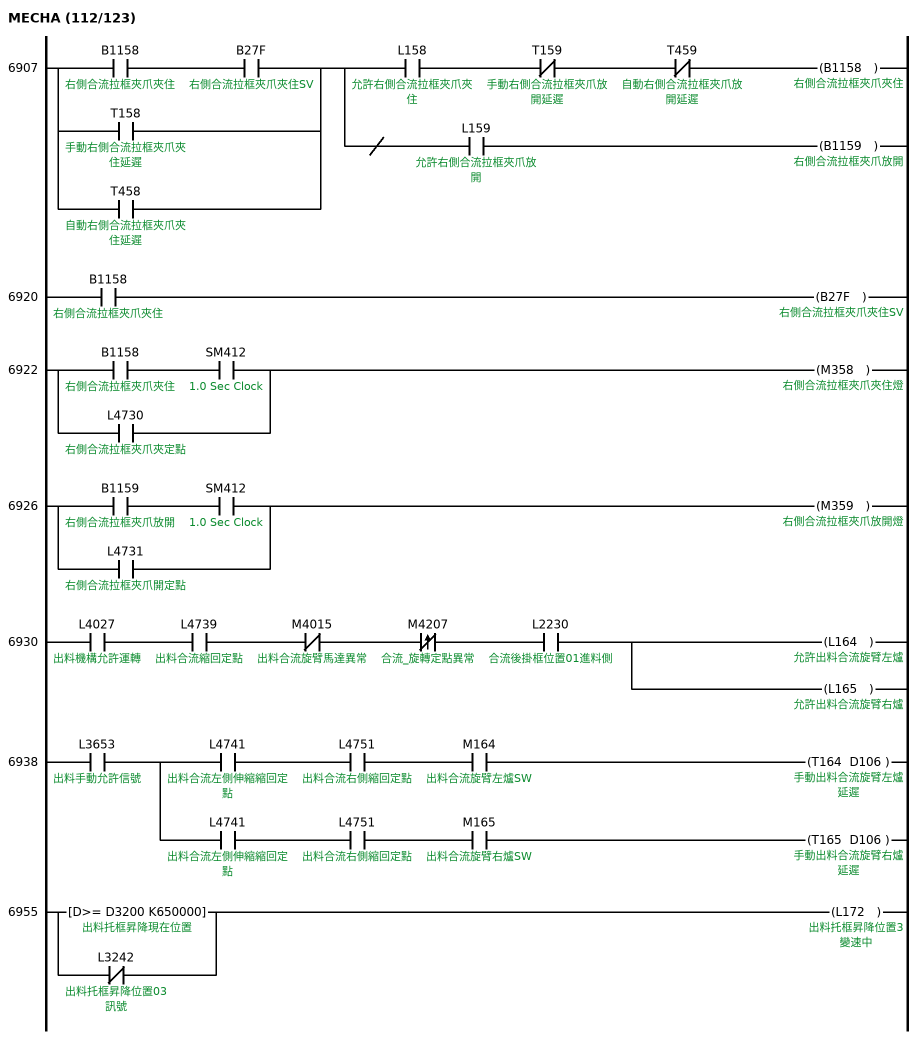
[picture p408: ladder of MECHA, rungs at steps 6907 to 6955]
6907  LD      B1158  ; 右側合流拉框夾爪夾住
      AND     B27F  ; 右側合流拉框夾爪夾住SV
      OR      T158  ; 手動右側合流拉框夾爪夾住延遲
      OR      T458  ; 自動右側合流拉框夾爪夾住延遲
      MPS
      AND     L158  ; 允許右側合流拉框夾爪夾住
      ANI     T159  ; 手動右側合流拉框夾爪放開延遲
      ANI     T459  ; 自動右側合流拉框夾爪放開延遲
      OUT     B1158  ; 右側合流拉框夾爪夾住
      MPP
      INV
      AND     L159  ; 允許右側合流拉框夾爪放開
      OUT     B1159  ; 右側合流拉框夾爪放開
6920  LD      B1158  ; 右側合流拉框夾爪夾住
      OUT     B27F  ; 右側合流拉框夾爪夾住SV
6922  LD      B1158  ; 右側合流拉框夾爪夾住
      AND     SM412  ; 1.0 Sec Clock
      OR      L4730  ; 右側合流拉框夾爪夾定點
      OUT     M358  ; 右側合流拉框夾爪夾住燈
6926  LD      B1159  ; 右側合流拉框夾爪放開
      AND     SM412  ; 1.0 Sec Clock
      OR      L4731  ; 右側合流拉框夾爪開定點
      OUT     M359  ; 右側合流拉框夾爪放開燈
6930  LD      L4027  ; 出料機構允許運轉
      AND     L4739  ; 出料合流縮回定點
      ANI     M4015  ; 出料合流旋臂馬達異常
      ANDPI   M4207  ; 合流_旋轉定點異常
      AND     L2230  ; 合流後掛框位置01進料側
      OUT     L164  ; 允許出料合流旋臂左爐
      OUT     L165  ; 允許出料合流旋臂右爐
6938  LD      L3653  ; 出料手動允許信號
      MPS
      AND     L4741  ; 出料合流左側伸縮縮回定點
      AND     L4751  ; 出料合流右側縮回定點
      AND     M164  ; 出料合流旋臂左爐SW
      OUT     T164 D106  ; 手動出料合流旋臂左爐延遲
      MPP
      AND     L4741  ; 出料合流左側伸縮縮回定點
      AND     L4751  ; 出料合流右側縮回定點
      AND     M165  ; 出料合流旋臂右爐SW
      OUT     T165 D106  ; 手動出料合流旋臂右爐延遲
6955  LDD>=   D3200 K650000  ; 出料托框昇降現在位置
      ORI     L3242  ; 出料托框昇降位置03 訊號
      OUT     L172  ; 出料托框昇降位置3 變速中
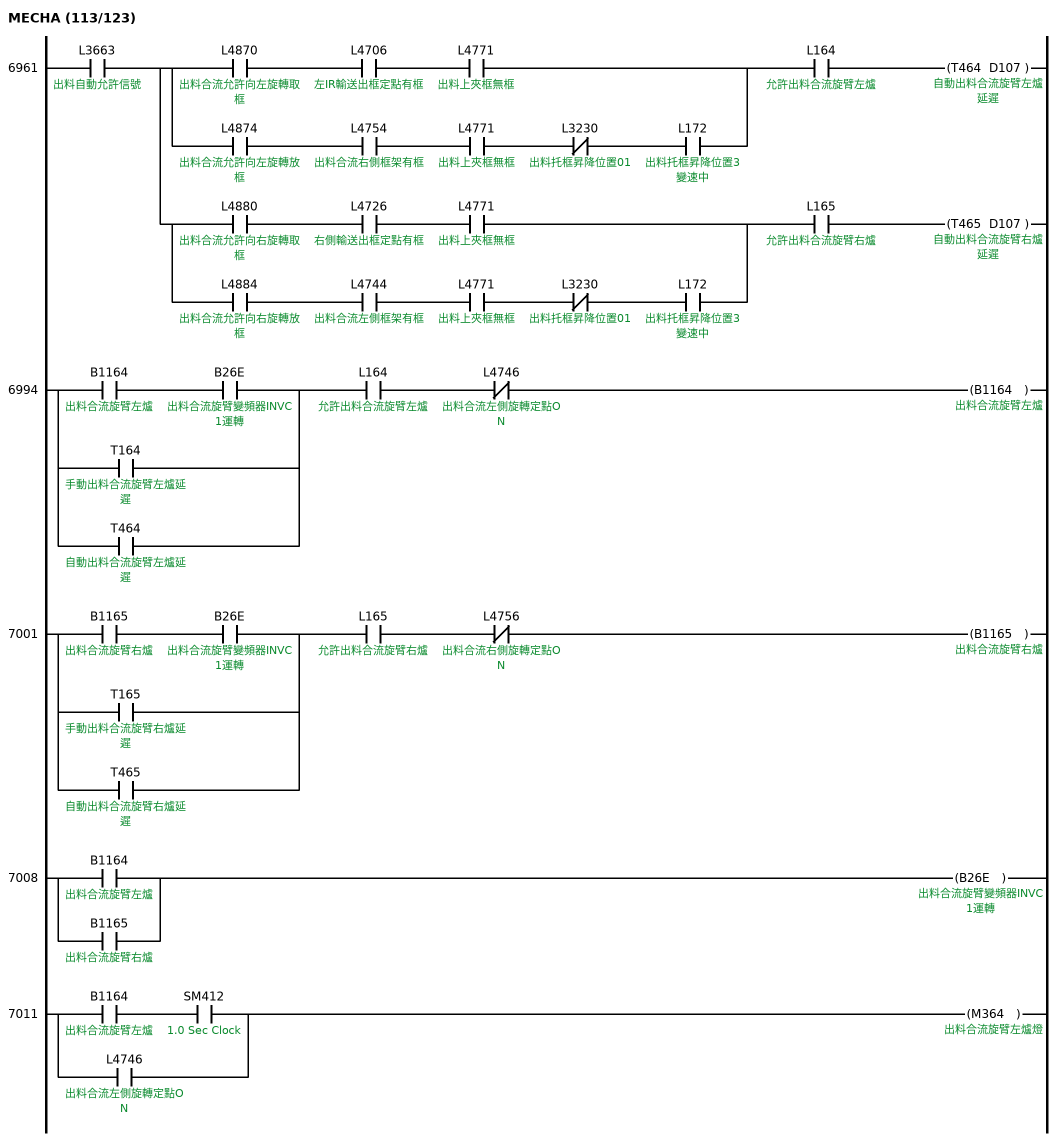
6961  LD      L3663  ; 出料自動允許信號
      MPS
      LD      L4870  ; 出料合流允許向左旋轉取框
      AND     L4706  ; 左IR輸送出框定點有框
      AND     L4771  ; 出料上夾框無框
      LD      L4874  ; 出料合流允許向左旋轉放框
      AND     L4754  ; 出料合流右側框架有框
      AND     L4771  ; 出料上夾框無框
      ANI     L3230  ; 出料托框昇降位置01
      AND     L172  ; 出料托框昇降位置3 變速中
      ORB
      ANB
      AND     L164  ; 允許出料合流旋臂左爐
      OUT     T464 D107  ; 自動出料合流旋臂左爐延遲
      MPP
      LD      L4880  ; 出料合流允許向右旋轉取框
      AND     L4726  ; 右側輸送出框定點有框
      AND     L4771  ; 出料上夾框無框
      LD      L4884  ; 出料合流允許向右旋轉放框
      AND     L4744  ; 出料合流左側框架有框
      AND     L4771  ; 出料上夾框無框
      ANI     L3230  ; 出料托框昇降位置01
      AND     L172  ; 出料托框昇降位置3 變速中
      ORB
      ANB
      AND     L165  ; 允許出料合流旋臂右爐
      OUT     T465 D107  ; 自動出料合流旋臂右爐延遲
6994  LD      B1164  ; 出料合流旋臂左爐
      AND     B26E  ; 出料合流旋臂變頻器INVC1運轉
      OR      T164  ; 手動出料合流旋臂左爐延遲
      OR      T464  ; 自動出料合流旋臂左爐延遲
      AND     L164  ; 允許出料合流旋臂左爐
      ANI     L4746  ; 出料合流左側旋轉定點ON
      OUT     B1164  ; 出料合流旋臂左爐
7001  LD      B1165  ; 出料合流旋臂右爐
      AND     B26E  ; 出料合流旋臂變頻器INVC1運轉
      OR      T165  ; 手動出料合流旋臂右爐延遲
      OR      T465  ; 自動出料合流旋臂右爐延遲
      AND     L165  ; 允許出料合流旋臂右爐
      ANI     L4756  ; 出料合流右側旋轉定點ON
      OUT     B1165  ; 出料合流旋臂右爐
7008  LD      B1164  ; 出料合流旋臂左爐
      OR      B1165  ; 出料合流旋臂右爐
      OUT     B26E  ; 出料合流旋臂變頻器INVC1運轉
7011  LD      B1164  ; 出料合流旋臂左爐
      AND     SM412  ; 1.0 Sec Clock
      OR      L4746  ; 出料合流左側旋轉定點ON
      OUT     M364  ; 出料合流旋臂左爐燈
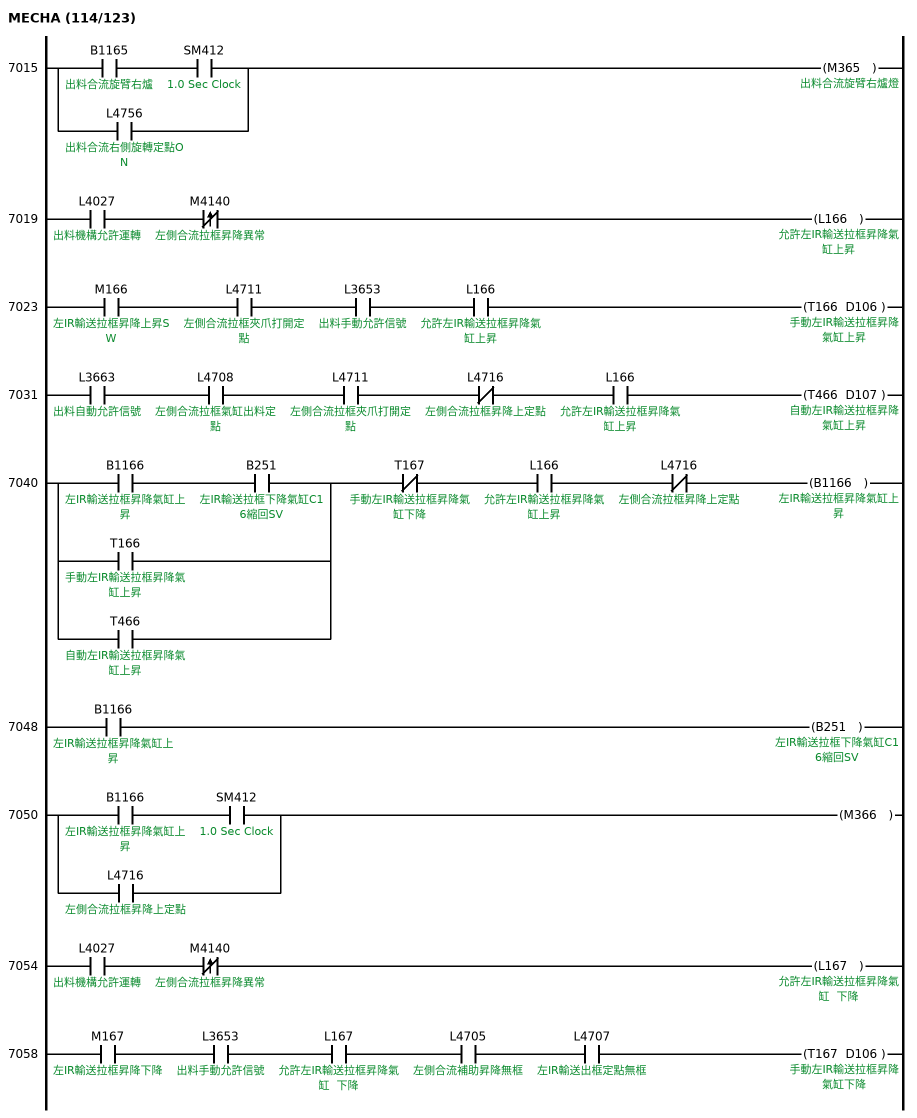
7015  LD      B1165  ; 出料合流旋臂右爐
      AND     SM412  ; 1.0 Sec Clock
      OR      L4756  ; 出料合流右側旋轉定點ON
      OUT     M365  ; 出料合流旋臂右爐燈
7019  LD      L4027  ; 出料機構允許運轉
      ANDPI   M4140  ; 左側合流拉框昇降異常
      OUT     L166  ; 允許左IR輸送拉框昇降氣缸上昇
7023  LD      M166  ; 左IR輸送拉框昇降上昇SW
      AND     L4711  ; 左側合流拉框夾爪打開定點
      AND     L3653  ; 出料手動允許信號
      AND     L166  ; 允許左IR輸送拉框昇降氣缸上昇
      OUT     T166 D106  ; 手動左IR輸送拉框昇降氣缸上昇
7031  LD      L3663  ; 出料自動允許信號
      AND     L4708  ; 左側合流拉框氣缸出料定點
      AND     L4711  ; 左側合流拉框夾爪打開定點
      ANI     L4716  ; 左側合流拉框昇降上定點
      AND     L166  ; 允許左IR輸送拉框昇降氣缸上昇
      OUT     T466 D107  ; 自動左IR輸送拉框昇降氣缸上昇
7040  LD      B1166  ; 左IR輸送拉框昇降氣缸上昇
      AND     B251  ; 左IR輸送拉框下降氣缸C16縮回SV
      OR      T166  ; 手動左IR輸送拉框昇降氣缸上昇
      OR      T466  ; 自動左IR輸送拉框昇降氣缸上昇
      ANI     T167  ; 手動左IR輸送拉框昇降氣缸下降
      AND     L166  ; 允許左IR輸送拉框昇降氣缸上昇
      ANI     L4716  ; 左側合流拉框昇降上定點
      OUT     B1166  ; 左IR輸送拉框昇降氣缸上昇
7048  LD      B1166  ; 左IR輸送拉框昇降氣缸上昇
      OUT     B251  ; 左IR輸送拉框下降氣缸C16縮回SV
7050  LD      B1166  ; 左IR輸送拉框昇降氣缸上昇
      AND     SM412  ; 1.0 Sec Clock
      OR      L4716  ; 左側合流拉框昇降上定點
      OUT     M366
7054  LD      L4027  ; 出料機構允許運轉
      ANDPI   M4140  ; 左側合流拉框昇降異常
      OUT     L167  ; 允許左IR輸送拉框昇降氣缸  下降
7058  LD      M167  ; 左IR輸送拉框昇降下降
      AND     L3653  ; 出料手動允許信號
      AND     L167  ; 允許左IR輸送拉框昇降氣缸  下降
      AND     L4705  ; 左側合流補助昇降無框
      AND     L4707  ; 左IR輸送出框定點無框
      OUT     T167 D106  ; 手動左IR輸送拉框昇降氣缸下降
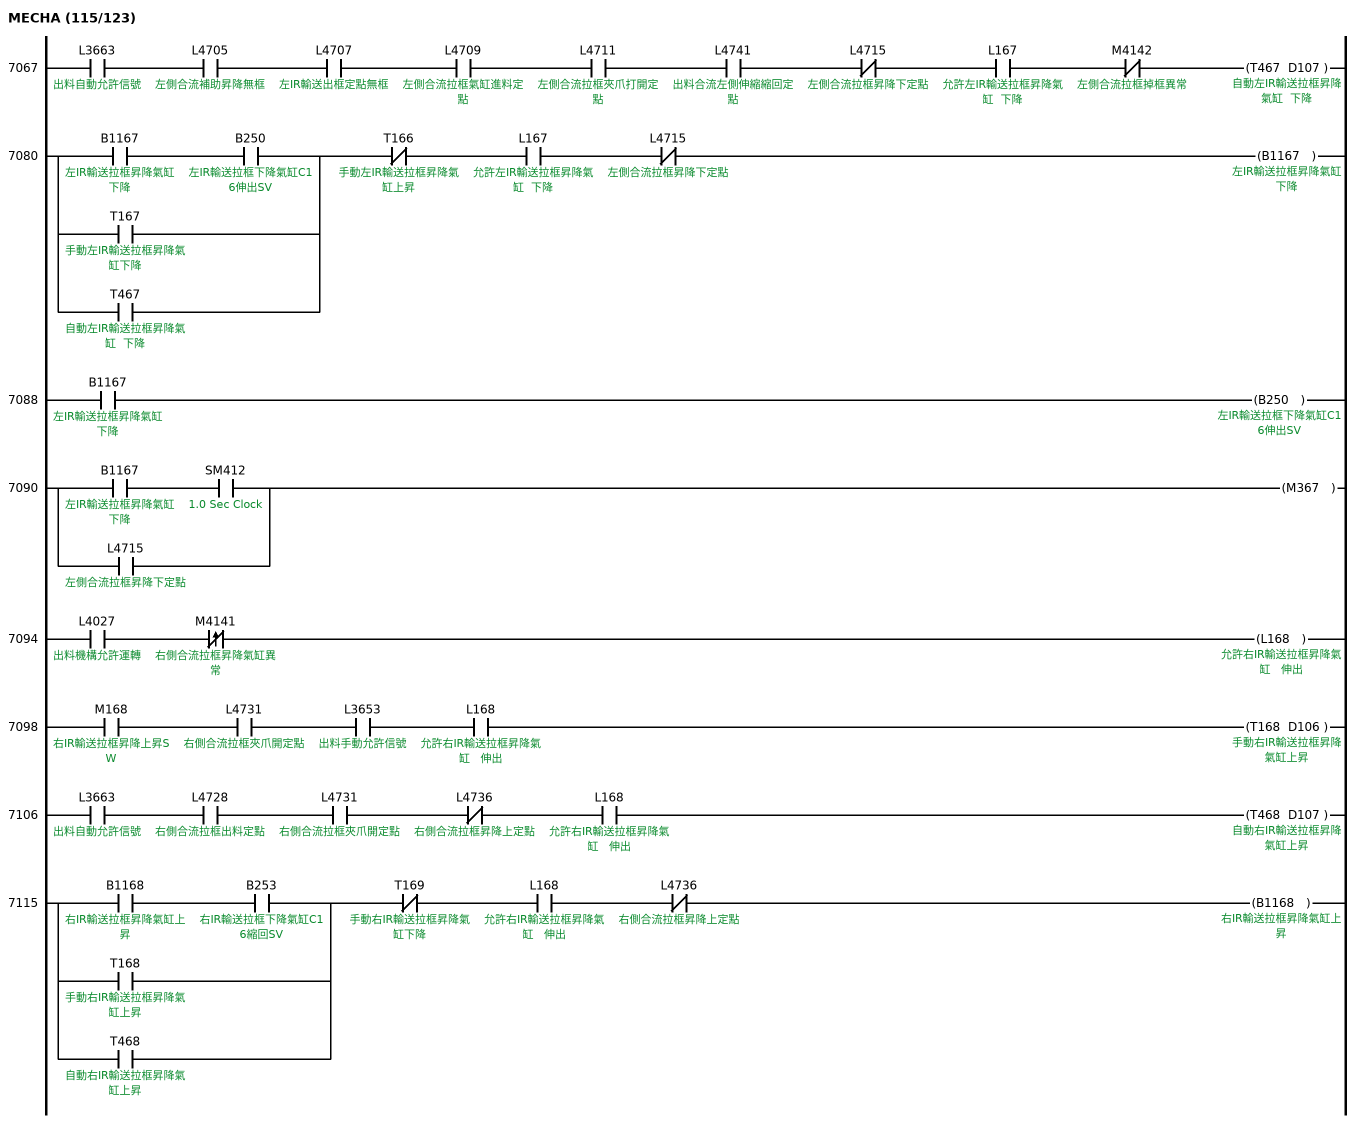
7067  LD      L3663  ; 出料自動允許信號
      AND     L4705  ; 左側合流補助昇降無框
      AND     L4707  ; 左IR輸送出框定點無框
      AND     L4709  ; 左側合流拉框氣缸進料定點
      AND     L4711  ; 左側合流拉框夾爪打開定點
      AND     L4741  ; 出料合流左側伸縮縮回定點
      ANI     L4715  ; 左側合流拉框昇降下定點
      AND     L167  ; 允許左IR輸送拉框昇降氣缸  下降
      ANI     M4142  ; 左側合流拉框掉框異常
      OUT     T467 D107  ; 自動左IR輸送拉框昇降氣缸  下降
7080  LD      B1167  ; 左IR輸送拉框昇降氣缸  下降
      AND     B250  ; 左IR輸送拉框下降氣缸C16伸出SV
      OR      T167  ; 手動左IR輸送拉框昇降氣缸下降
      OR      T467  ; 自動左IR輸送拉框昇降氣缸  下降
      ANI     T166  ; 手動左IR輸送拉框昇降氣缸上昇
      AND     L167  ; 允許左IR輸送拉框昇降氣缸  下降
      ANI     L4715  ; 左側合流拉框昇降下定點
      OUT     B1167  ; 左IR輸送拉框昇降氣缸  下降
7088  LD      B1167  ; 左IR輸送拉框昇降氣缸  下降
      OUT     B250  ; 左IR輸送拉框下降氣缸C16伸出SV
7090  LD      B1167  ; 左IR輸送拉框昇降氣缸  下降
      AND     SM412  ; 1.0 Sec Clock
      OR      L4715  ; 左側合流拉框昇降下定點
      OUT     M367
7094  LD      L4027  ; 出料機構允許運轉
      ANDPI   M4141  ; 右側合流拉框昇降氣缸異常
      OUT     L168  ; 允許右IR輸送拉框昇降氣缸   伸出
7098  LD      M168  ; 右IR輸送拉框昇降上昇SW
      AND     L4731  ; 右側合流拉框夾爪開定點
      AND     L3653  ; 出料手動允許信號
      AND     L168  ; 允許右IR輸送拉框昇降氣缸   伸出
      OUT     T168 D106  ; 手動右IR輸送拉框昇降氣缸上昇
7106  LD      L3663  ; 出料自動允許信號
      AND     L4728  ; 右側合流拉框出料定點
      AND     L4731  ; 右側合流拉框夾爪開定點
      ANI     L4736  ; 右側合流拉框昇降上定點
      AND     L168  ; 允許右IR輸送拉框昇降氣缸   伸出
      OUT     T468 D107  ; 自動右IR輸送拉框昇降氣缸上昇
7115  LD      B1168  ; 右IR輸送拉框昇降氣缸上昇
      AND     B253  ; 右IR輸送拉框下降氣缸C16縮回SV
      OR      T168  ; 手動右IR輸送拉框昇降氣缸上昇
      OR      T468  ; 自動右IR輸送拉框昇降氣缸上昇
      ANI     T169  ; 手動右IR輸送拉框昇降氣缸下降
      AND     L168  ; 允許右IR輸送拉框昇降氣缸   伸出
      ANI     L4736  ; 右側合流拉框昇降上定點
      OUT     B1168  ; 右IR輸送拉框昇降氣缸上昇
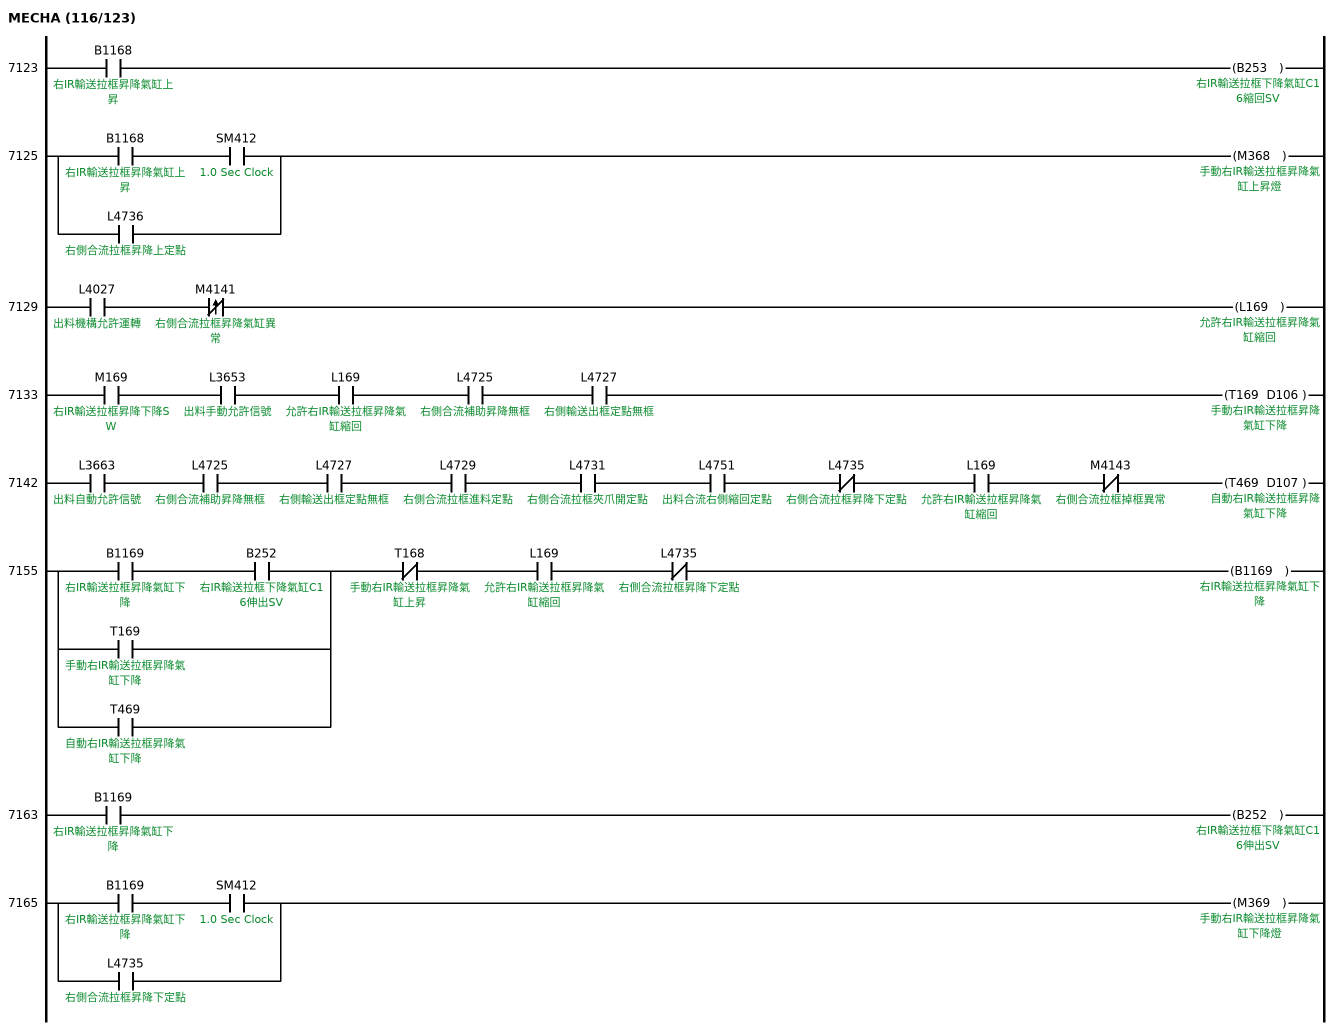
7123  LD      B1168  ; 右IR輸送拉框昇降氣缸上昇
      OUT     B253  ; 右IR輸送拉框下降氣缸C16縮回SV
7125  LD      B1168  ; 右IR輸送拉框昇降氣缸上昇
      AND     SM412  ; 1.0 Sec Clock
      OR      L4736  ; 右側合流拉框昇降上定點
      OUT     M368  ; 手動右IR輸送拉框昇降氣缸上昇燈
7129  LD      L4027  ; 出料機構允許運轉
      ANDPI   M4141  ; 右側合流拉框昇降氣缸異常
      OUT     L169  ; 允許右IR輸送拉框昇降氣缸縮回
7133  LD      M169  ; 右IR輸送拉框昇降下降SW
      AND     L3653  ; 出料手動允許信號
      AND     L169  ; 允許右IR輸送拉框昇降氣缸縮回
      AND     L4725  ; 右側合流補助昇降無框
      AND     L4727  ; 右側輸送出框定點無框
      OUT     T169 D106  ; 手動右IR輸送拉框昇降氣缸下降
7142  LD      L3663  ; 出料自動允許信號
      AND     L4725  ; 右側合流補助昇降無框
      AND     L4727  ; 右側輸送出框定點無框
      AND     L4729  ; 右側合流拉框進料定點
      AND     L4731  ; 右側合流拉框夾爪開定點
      AND     L4751  ; 出料合流右側縮回定點
      ANI     L4735  ; 右側合流拉框昇降下定點
      AND     L169  ; 允許右IR輸送拉框昇降氣缸縮回
      ANI     M4143  ; 右側合流拉框掉框異常
      OUT     T469 D107  ; 自動右IR輸送拉框昇降氣缸下降
7155  LD      B1169  ; 右IR輸送拉框昇降氣缸下降
      AND     B252  ; 右IR輸送拉框下降氣缸C16伸出SV
      OR      T169  ; 手動右IR輸送拉框昇降氣缸下降
      OR      T469  ; 自動右IR輸送拉框昇降氣缸下降
      ANI     T168  ; 手動右IR輸送拉框昇降氣缸上昇
      AND     L169  ; 允許右IR輸送拉框昇降氣缸縮回
      ANI     L4735  ; 右側合流拉框昇降下定點
      OUT     B1169  ; 右IR輸送拉框昇降氣缸下降
7163  LD      B1169  ; 右IR輸送拉框昇降氣缸下降
      OUT     B252  ; 右IR輸送拉框下降氣缸C16伸出SV
7165  LD      B1169  ; 右IR輸送拉框昇降氣缸下降
      AND     SM412  ; 1.0 Sec Clock
      OR      L4735  ; 右側合流拉框昇降下定點
      OUT     M369  ; 手動右IR輸送拉框昇降氣缸下降燈
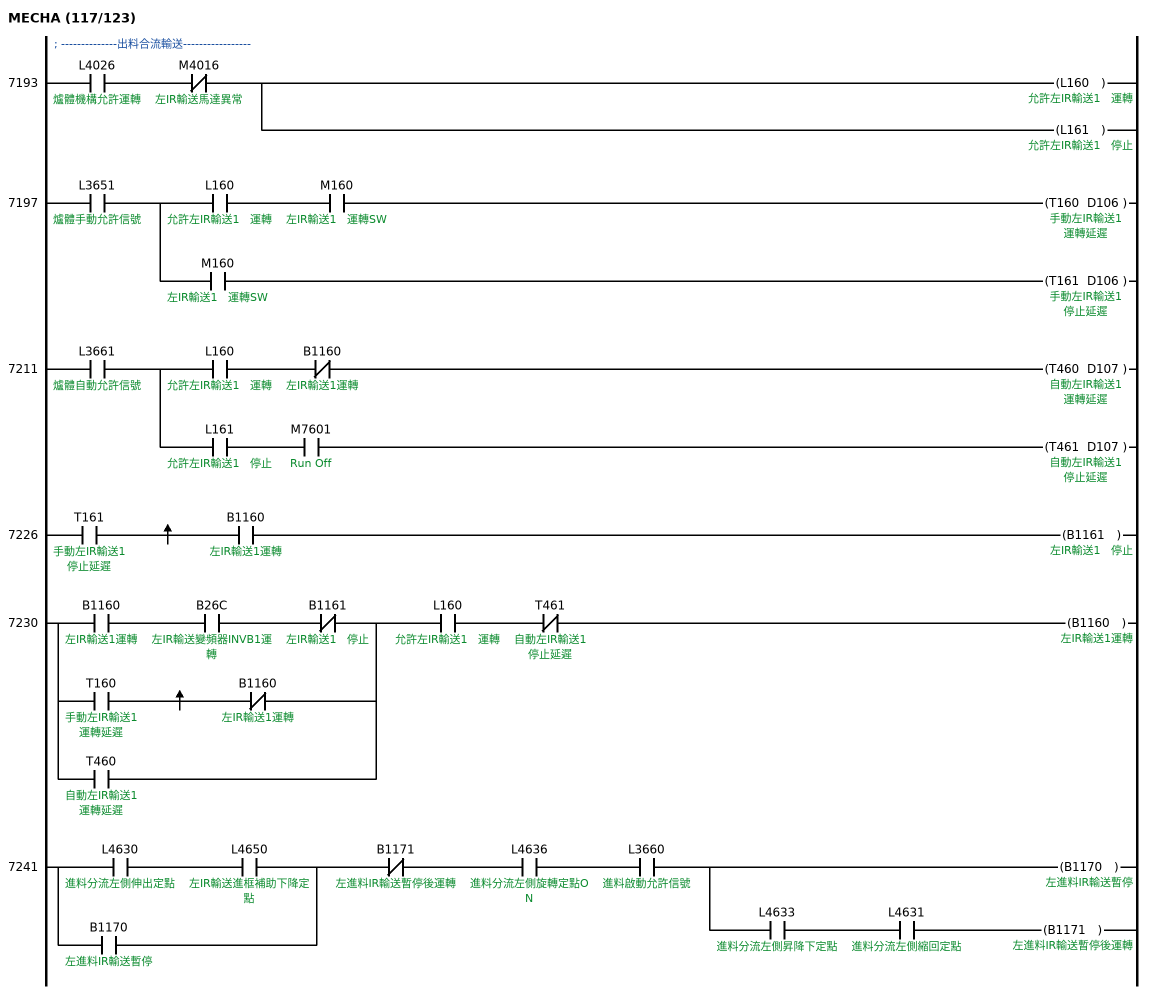
; --------------出料合流輸送-----------------
7193  LD      L4026  ; 爐體機構允許運轉
      ANI     M4016  ; 左IR輸送馬達異常
      OUT     L160  ; 允許左IR輸送1   運轉
      OUT     L161  ; 允許左IR輸送1   停止
7197  LD      L3651  ; 爐體手動允許信號
      MPS
      AND     L160  ; 允許左IR輸送1   運轉
      AND     M160  ; 左IR輸送1   運轉SW
      OUT     T160 D106  ; 手動左IR輸送1   運轉延遲
      MPP
      AND     M160  ; 左IR輸送1   運轉SW
      OUT     T161 D106  ; 手動左IR輸送1   停止延遲
7211  LD      L3661  ; 爐體自動允許信號
      MPS
      AND     L160  ; 允許左IR輸送1   運轉
      ANI     B1160  ; 左IR輸送1運轉
      OUT     T460 D107  ; 自動左IR輸送1   運轉延遲
      MPP
      AND     L161  ; 允許左IR輸送1   停止
      AND     M7601  ; Run Off
      OUT     T461 D107  ; 自動左IR輸送1   停止延遲
7226  LD      T161  ; 手動左IR輸送1   停止延遲
      MEP
      AND     B1160  ; 左IR輸送1運轉
      OUT     B1161  ; 左IR輸送1   停止
7230  LD      B1160  ; 左IR輸送1運轉
      AND     B26C  ; 左IR輸送變頻器INVB1運轉
      ANI     B1161  ; 左IR輸送1   停止
      LD      T160  ; 手動左IR輸送1   運轉延遲
      MEP
      ANI     B1160  ; 左IR輸送1運轉
      ORB
      OR      T460  ; 自動左IR輸送1   運轉延遲
      AND     L160  ; 允許左IR輸送1   運轉
      ANI     T461  ; 自動左IR輸送1   停止延遲
      OUT     B1160  ; 左IR輸送1運轉
7241  LD      L4630  ; 進料分流左側伸出定點
      AND     L4650  ; 左IR輸送進框補助下降定點
      OR      B1170  ; 左進料IR輸送暫停
      ANI     B1171  ; 左進料IR輸送暫停後運轉
      AND     L4636  ; 進料分流左側旋轉定點ON
      AND     L3660  ; 進料啟動允許信號
      OUT     B1170  ; 左進料IR輸送暫停
      AND     L4633  ; 進料分流左側昇降下定點
      AND     L4631  ; 進料分流左側縮回定點
      OUT     B1171  ; 左進料IR輸送暫停後運轉
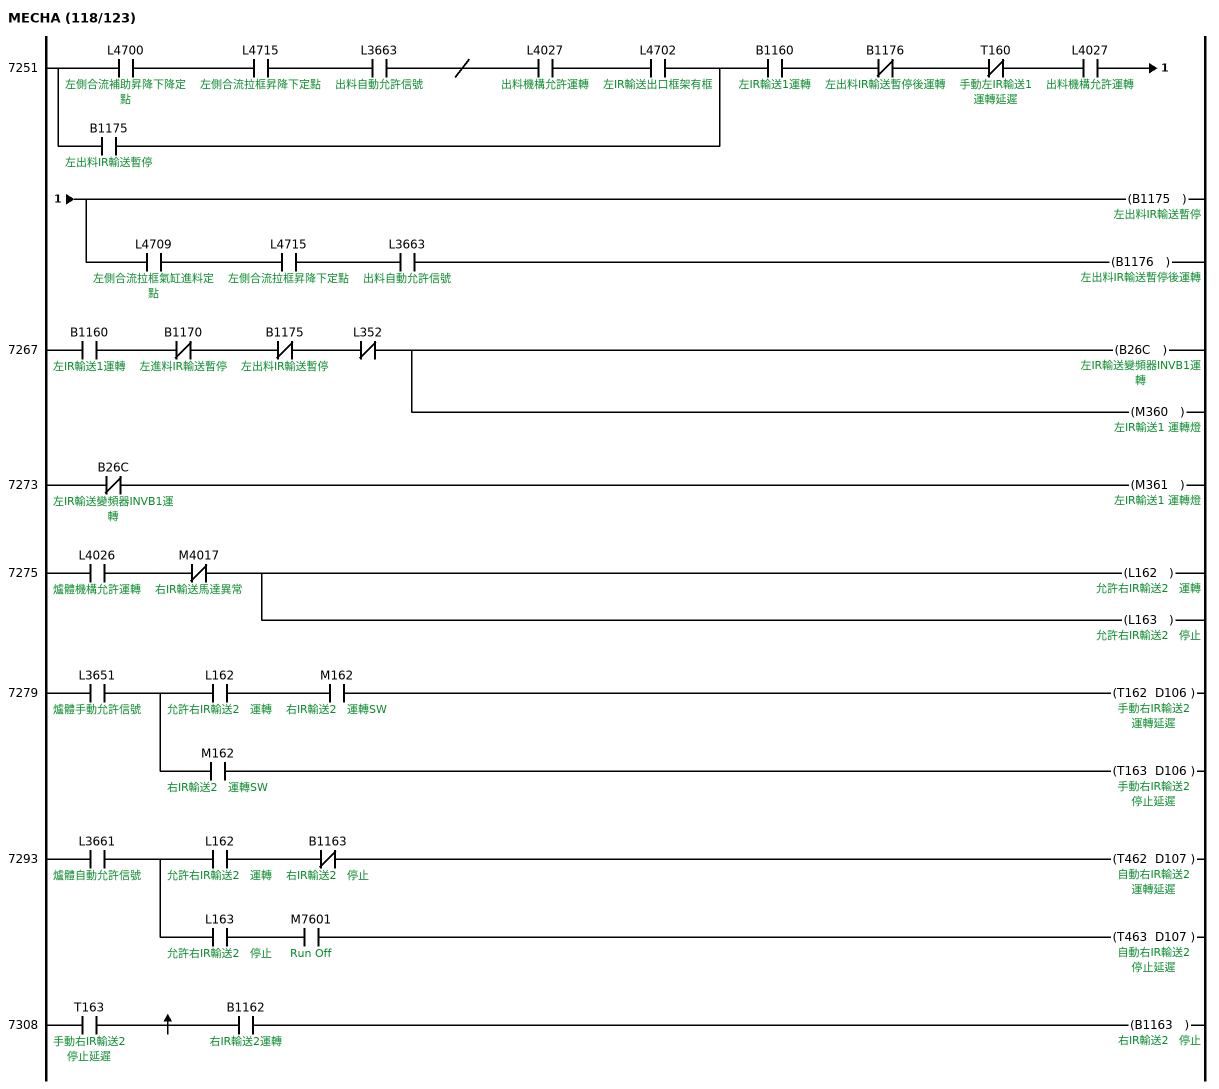
7251  LD      L4700  ; 左側合流補助昇降下降定點
      AND     L4715  ; 左側合流拉框昇降下定點
      AND     L3663  ; 出料自動允許信號
      INV
      AND     L4027  ; 出料機構允許運轉
      AND     L4702  ; 左IR輸送出口框架有框
      OR      B1175  ; 左出料IR輸送暫停
      AND     B1160  ; 左IR輸送1運轉
      ANI     B1176  ; 左出料IR輸送暫停後運轉
      ANI     T160  ; 手動左IR輸送1   運轉延遲
      AND     L4027  ; 出料機構允許運轉
      OUT     B1175  ; 左出料IR輸送暫停
      AND     L4709  ; 左側合流拉框氣缸進料定點
      AND     L4715  ; 左側合流拉框昇降下定點
      AND     L3663  ; 出料自動允許信號
      OUT     B1176  ; 左出料IR輸送暫停後運轉
7267  LD      B1160  ; 左IR輸送1運轉
      ANI     B1170  ; 左進料IR輸送暫停
      ANI     B1175  ; 左出料IR輸送暫停
      ANI     L352
      OUT     B26C  ; 左IR輸送變頻器INVB1運轉
      OUT     M360  ; 左IR輸送1 運轉燈
7273  LDI     B26C  ; 左IR輸送變頻器INVB1運轉
      OUT     M361  ; 左IR輸送1 運轉燈
7275  LD      L4026  ; 爐體機構允許運轉
      ANI     M4017  ; 右IR輸送馬達異常
      OUT     L162  ; 允許右IR輸送2   運轉
      OUT     L163  ; 允許右IR輸送2   停止
7279  LD      L3651  ; 爐體手動允許信號
      MPS
      AND     L162  ; 允許右IR輸送2   運轉
      AND     M162  ; 右IR輸送2   運轉SW
      OUT     T162 D106  ; 手動右IR輸送2   運轉延遲
      MPP
      AND     M162  ; 右IR輸送2   運轉SW
      OUT     T163 D106  ; 手動右IR輸送2   停止延遲
7293  LD      L3661  ; 爐體自動允許信號
      MPS
      AND     L162  ; 允許右IR輸送2   運轉
      ANI     B1163  ; 右IR輸送2   停止
      OUT     T462 D107  ; 自動右IR輸送2   運轉延遲
      MPP
      AND     L163  ; 允許右IR輸送2   停止
      AND     M7601  ; Run Off
      OUT     T463 D107  ; 自動右IR輸送2   停止延遲
7308  LD      T163  ; 手動右IR輸送2   停止延遲
      MEP
      AND     B1162  ; 右IR輸送2運轉
      OUT     B1163  ; 右IR輸送2   停止
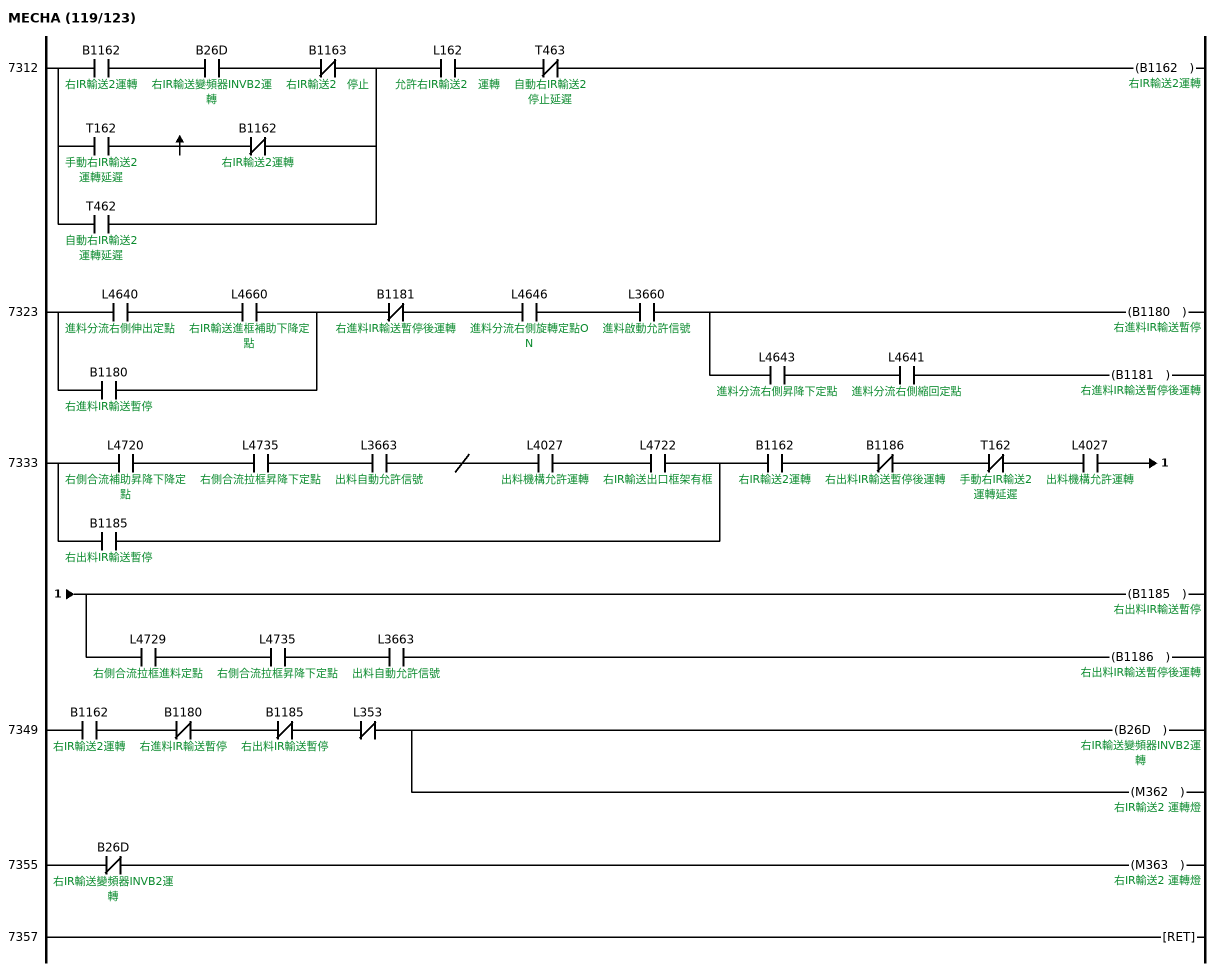
7312  LD      B1162  ; 右IR輸送2運轉
      AND     B26D  ; 右IR輸送變頻器INVB2運轉
      ANI     B1163  ; 右IR輸送2   停止
      LD      T162  ; 手動右IR輸送2   運轉延遲
      MEP
      ANI     B1162  ; 右IR輸送2運轉
      ORB
      OR      T462  ; 自動右IR輸送2   運轉延遲
      AND     L162  ; 允許右IR輸送2   運轉
      ANI     T463  ; 自動右IR輸送2   停止延遲
      OUT     B1162  ; 右IR輸送2運轉
7323  LD      L4640  ; 進料分流右側伸出定點
      AND     L4660  ; 右IR輸送進框補助下降定點
      OR      B1180  ; 右進料IR輸送暫停
      ANI     B1181  ; 右進料IR輸送暫停後運轉
      AND     L4646  ; 進料分流右側旋轉定點ON
      AND     L3660  ; 進料啟動允許信號
      OUT     B1180  ; 右進料IR輸送暫停
      AND     L4643  ; 進料分流右側昇降下定點
      AND     L4641  ; 進料分流右側縮回定點
      OUT     B1181  ; 右進料IR輸送暫停後運轉
7333  LD      L4720  ; 右側合流補助昇降下降定點
      AND     L4735  ; 右側合流拉框昇降下定點
      AND     L3663  ; 出料自動允許信號
      INV
      AND     L4027  ; 出料機構允許運轉
      AND     L4722  ; 右IR輸送出口框架有框
      OR      B1185  ; 右出料IR輸送暫停
      AND     B1162  ; 右IR輸送2運轉
      ANI     B1186  ; 右出料IR輸送暫停後運轉
      ANI     T162  ; 手動右IR輸送2   運轉延遲
      AND     L4027  ; 出料機構允許運轉
      OUT     B1185  ; 右出料IR輸送暫停
      AND     L4729  ; 右側合流拉框進料定點
      AND     L4735  ; 右側合流拉框昇降下定點
      AND     L3663  ; 出料自動允許信號
      OUT     B1186  ; 右出料IR輸送暫停後運轉
7349  LD      B1162  ; 右IR輸送2運轉
      ANI     B1180  ; 右進料IR輸送暫停
      ANI     B1185  ; 右出料IR輸送暫停
      ANI     L353
      OUT     B26D  ; 右IR輸送變頻器INVB2運轉
      OUT     M362  ; 右IR輸送2 運轉燈
7355  LDI     B26D  ; 右IR輸送變頻器INVB2運轉
      OUT     M363  ; 右IR輸送2 運轉燈
7357  RET
      P1071
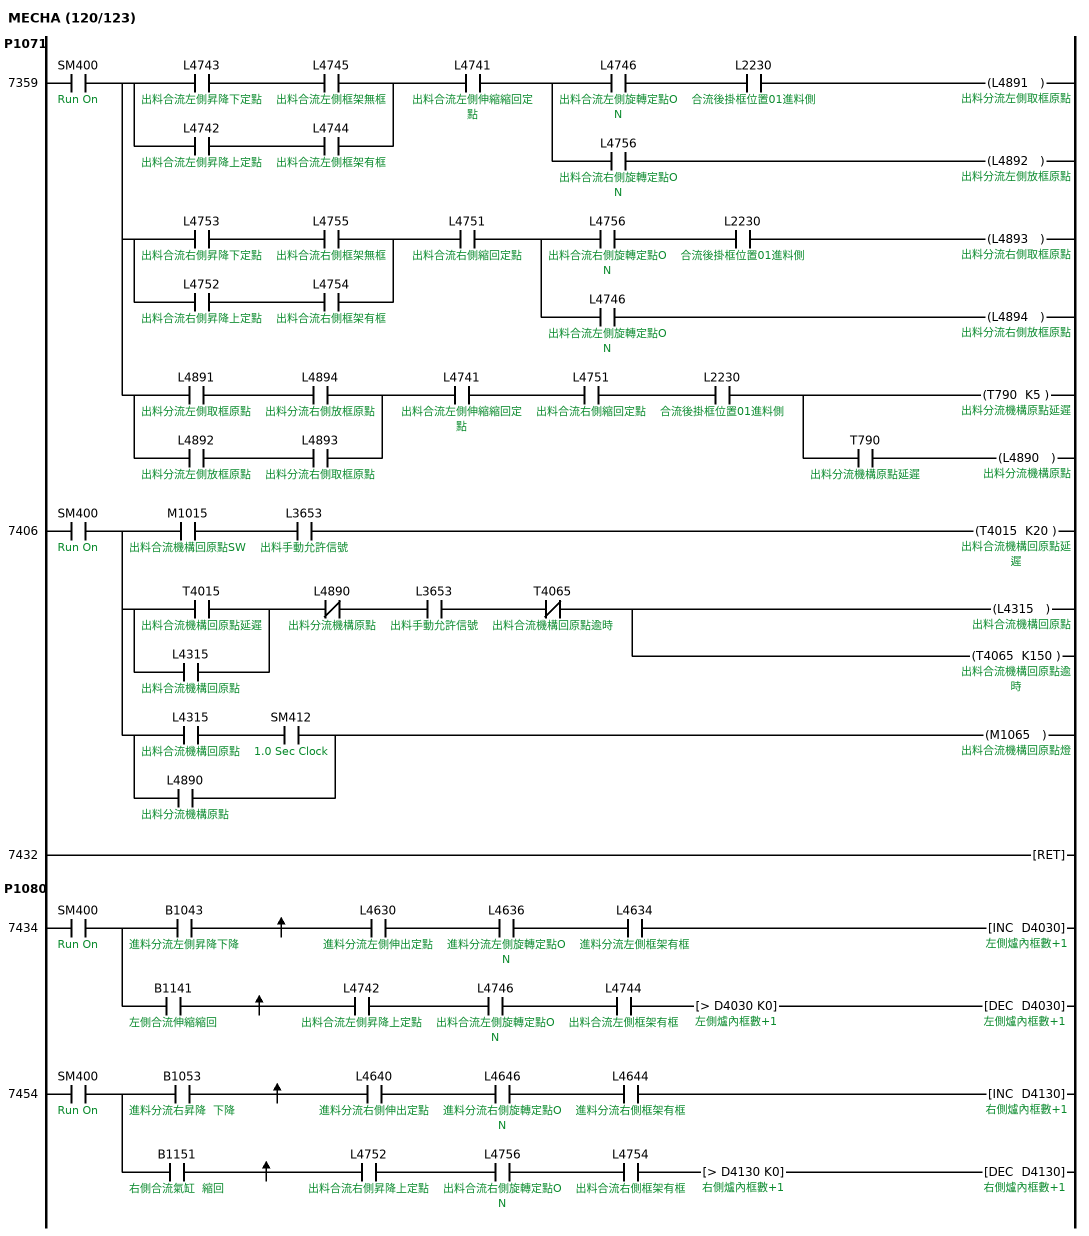
7359  LD      SM400  ; Run On
      MPS
      LD      L4743  ; 出料合流左側昇降下定點
      AND     L4745  ; 出料合流左側框架無框
      LD      L4742  ; 出料合流左側昇降上定點
      AND     L4744  ; 出料合流左側框架有框
      ORB
      ANB
      AND     L4741  ; 出料合流左側伸縮縮回定點
      MPS
      AND     L4746  ; 出料合流左側旋轉定點ON
      AND     L2230  ; 合流後掛框位置01進料側
      OUT     L4891  ; 出料分流左側取框原點
      MPP
      AND     L4756  ; 出料合流右側旋轉定點ON
      OUT     L4892  ; 出料分流左側放框原點
      MRD
      LD      L4753  ; 出料合流右側昇降下定點
      AND     L4755  ; 出料合流右側框架無框
      LD      L4752  ; 出料合流右側昇降上定點
      AND     L4754  ; 出料合流右側框架有框
      ORB
      ANB
      AND     L4751  ; 出料合流右側縮回定點
      MPS
      AND     L4756  ; 出料合流右側旋轉定點ON
      AND     L2230  ; 合流後掛框位置01進料側
      OUT     L4893  ; 出料分流右側取框原點
      MPP
      AND     L4746  ; 出料合流左側旋轉定點ON
      OUT     L4894  ; 出料分流右側放框原點
      MPP
      LD      L4891  ; 出料分流左側取框原點
      AND     L4894  ; 出料分流右側放框原點
      LD      L4892  ; 出料分流左側放框原點
      AND     L4893  ; 出料分流右側取框原點
      ORB
      ANB
      AND     L4741  ; 出料合流左側伸縮縮回定點
      AND     L4751  ; 出料合流右側縮回定點
      AND     L2230  ; 合流後掛框位置01進料側
      OUT     T790 K5  ; 出料分流機構原點延遲
      AND     T790  ; 出料分流機構原點延遲
      OUT     L4890  ; 出料分流機構原點
7406  LD      SM400  ; Run On
      MPS
      AND     M1015  ; 出料合流機構回原點SW
      AND     L3653  ; 出料手動允許信號
      OUT     T4015 K20  ; 出料合流機構回原點延遲
      MRD
      LD      T4015  ; 出料合流機構回原點延遲
      OR      L4315  ; 出料合流機構回原點
      ANB
      ANI     L4890  ; 出料分流機構原點
      AND     L3653  ; 出料手動允許信號
      ANI     T4065  ; 出料合流機構回原點逾時
      OUT     L4315  ; 出料合流機構回原點
      OUT     T4065 K150  ; 出料合流機構回原點逾時
      MPP
      LD      L4315  ; 出料合流機構回原點
      AND     SM412  ; 1.0 Sec Clock
      OR      L4890  ; 出料分流機構原點
      ANB
      OUT     M1065  ; 出料合流機構回原點燈
7432  RET
      P1080
7434  LD      SM400  ; Run On
      MPS
      AND     B1043  ; 進料分流左側昇降下降
      MEP
      AND     L4630  ; 進料分流左側伸出定點
      AND     L4636  ; 進料分流左側旋轉定點ON
      AND     L4634  ; 進料分流左側框架有框
      INC     D4030  ; 左側爐內框數+1
      MPP
      AND     B1141  ; 左側合流伸縮縮回
      MEP
      AND     L4742  ; 出料合流左側昇降上定點
      AND     L4746  ; 出料合流左側旋轉定點ON
      AND     L4744  ; 出料合流左側框架有框
      AND>    D4030 K0  ; 左側爐內框數+1
      DEC     D4030
7454  LD      SM400  ; Run On
      MPS
      AND     B1053  ; 進料分流右昇降  下降
      MEP
      AND     L4640  ; 進料分流右側伸出定點
      AND     L4646  ; 進料分流右側旋轉定點ON
      AND     L4644  ; 進料分流右側框架有框
      INC     D4130  ; 右側爐內框數+1
      MPP
      AND     B1151  ; 右側合流氣缸  縮回
      MEP
      AND     L4752  ; 出料合流右側昇降上定點
      AND     L4756  ; 出料合流右側旋轉定點ON
      AND     L4754  ; 出料合流右側框架有框
      AND>    D4130 K0  ; 右側爐內框數+1
      DEC     D4130
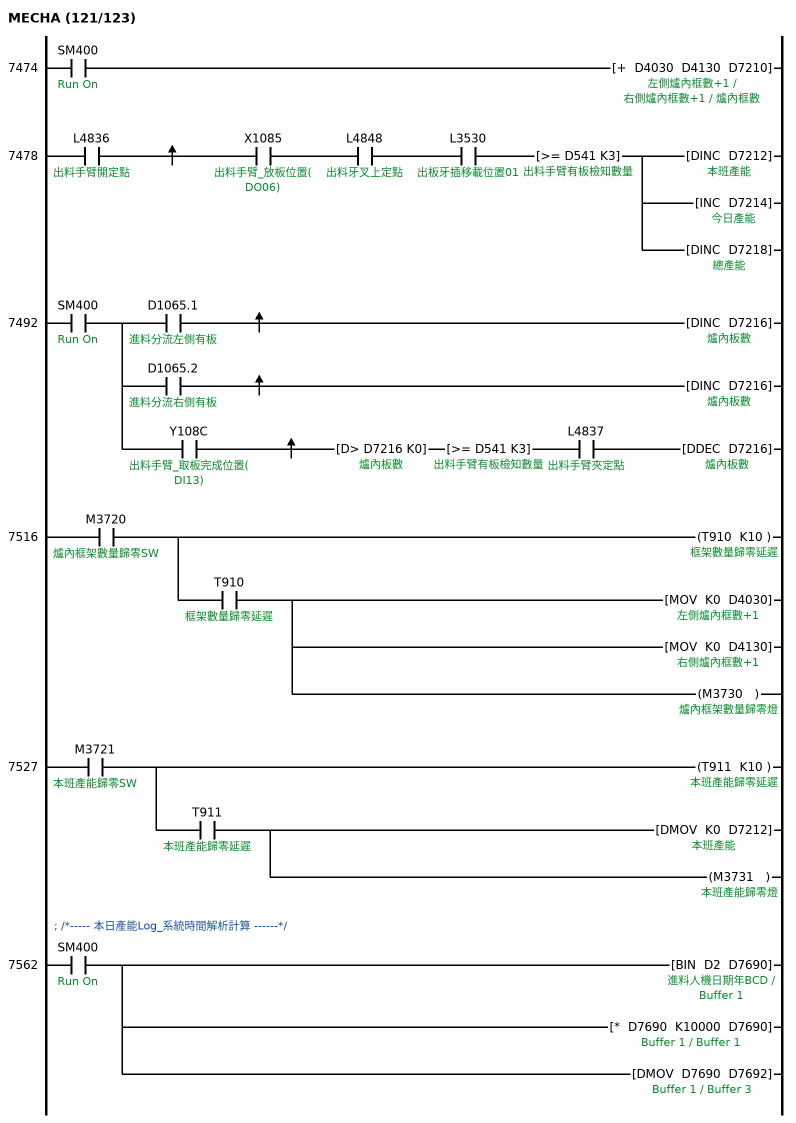
7474  LD      SM400  ; Run On
      +       D4030 D4130 D7210  ; 爐內框數
7478  LD      L4836  ; 出料手臂開定點
      MEP
      AND     X1085  ; 出料手臂_放板位置(DO06)
      AND     L4848  ; 出料牙叉上定點
      AND     L3530  ; 出板牙插移載位置01
      AND>=   D541 K3  ; 出料手臂有板檢知數量
      DINC    D7212  ; 本班產能
      INC     D7214  ; 今日產能
      DINC    D7218  ; 總產能
7492  LD      SM400  ; Run On
      MPS
      AND     D1065.1  ; 進料分流左側有板
      MEP
      DINC    D7216  ; 爐內板數
      MRD
      AND     D1065.2  ; 進料分流右側有板
      MEP
      DINC    D7216
      MPP
      AND     Y108C  ; 出料手臂_取板完成位置(DI13)
      MEP
      ANDD>   D7216 K0  ; 爐內板數
      AND>=   D541 K3  ; 出料手臂有板檢知數量
      AND     L4837  ; 出料手臂夾定點
      DDEC    D7216
7516  LD      M3720  ; 爐內框架數量歸零SW
      OUT     T910 K10  ; 框架數量歸零延遲
      AND     T910  ; 框架數量歸零延遲
      MOV     K0 D4030
      MOV     K0 D4130
      OUT     M3730  ; 爐內框架數量歸零燈
7527  LD      M3721  ; 本班產能歸零SW
      OUT     T911 K10  ; 本班產能歸零延遲
      AND     T911  ; 本班產能歸零延遲
      DMOV    K0 D7212
      OUT     M3731  ; 本班產能歸零燈
; /*----- 本日產能Log_系統時間解析計算 ------*/
7562  LD      SM400  ; Run On
      BIN     D2 D7690  ; 進料人機日期年BCD / Buffer 1
      *       D7690 K10000 D7690
      DMOV    D7690 D7692  ; Buffer 3
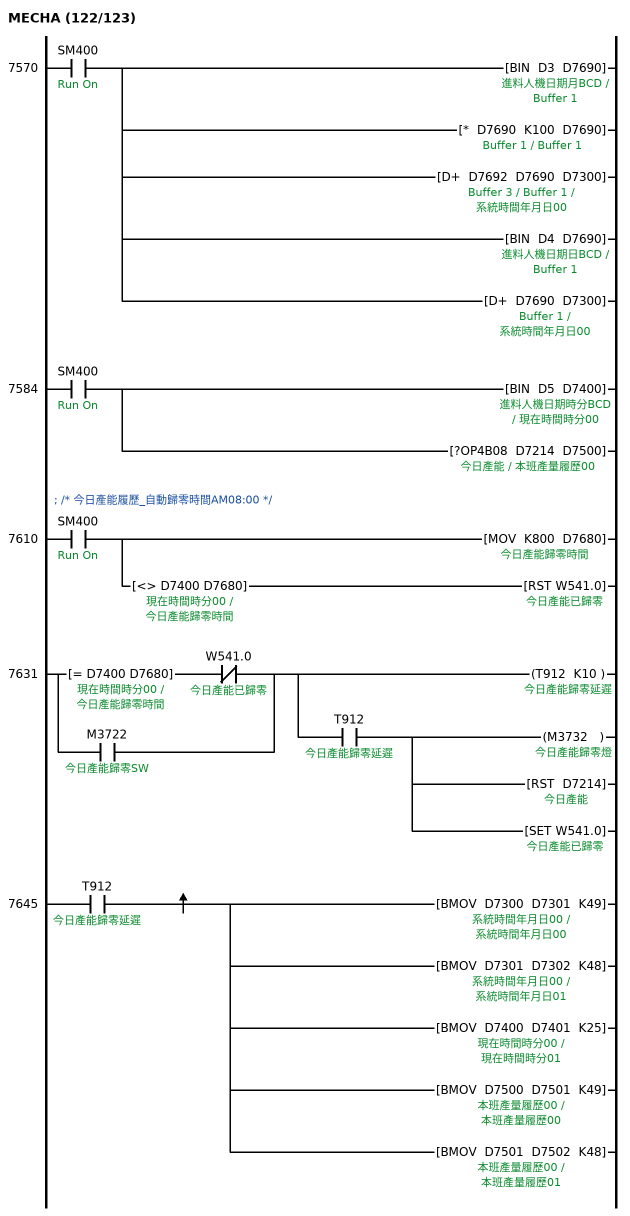
7570  LD      SM400  ; Run On
      BIN     D3 D7690  ; 進料人機日期月BCD
      *       D7690 K100 D7690
      D+      D7692 D7690 D7300  ; 系統時間年月日00
      BIN     D4 D7690  ; 進料人機日期日BCD
      D+      D7690 D7300
7584  LD      SM400  ; Run On
      BIN     D5 D7400  ; 進料人機日期時分BCD / 現在時間時分00
      ?OP4B08 D7214 D7500  ; 本班產量履歷00
; /* 今日產能履歷_自動歸零時間AM08:00 */
7610  LD      SM400  ; Run On
      MOV     K800 D7680  ; 今日產能歸零時間
        [note] 今日產能歸零時間_AM08:00
      AND<>   D7400 D7680  ; 現在時間時分00 / 今日產能歸零時間
      RST     W541.0  ; 今日產能已歸零
7631  LD=     D7400 D7680  ; 現在時間時分00 / 今日產能歸零時間
      ANI     W541.0  ; 今日產能已歸零
      OR      M3722  ; 今日產能歸零SW
      OUT     T912 K10  ; 今日產能歸零延遲
      AND     T912  ; 今日產能歸零延遲
      OUT     M3732  ; 今日產能歸零燈
      RST     D7214  ; 今日產能
      SET     W541.0  ; 今日產能已歸零
7645  LD      T912  ; 今日產能歸零延遲
      MEP
      BMOV    D7300 D7301 K49  ; 系統時間年月日00
      BMOV    D7301 D7302 K48  ; 系統時間年月日01
      BMOV    D7400 D7401 K25  ; 現在時間時分01
      BMOV    D7500 D7501 K49  ; 本班產量履歷00
      BMOV    D7501 D7502 K48  ; 本班產量履歷01
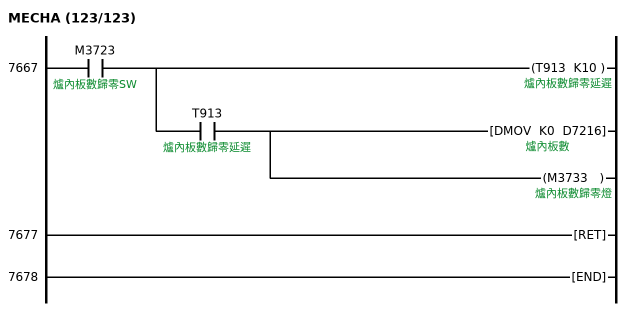
7667  LD      M3723  ; 爐內板數歸零SW
      OUT     T913 K10  ; 爐內板數歸零延遲
      AND     T913  ; 爐內板數歸零延遲
      DMOV    K0 D7216
      OUT     M3733  ; 爐內板數歸零燈
7677  RET
7678  END
END_PROGRAM

PROGRAM ORIGIN
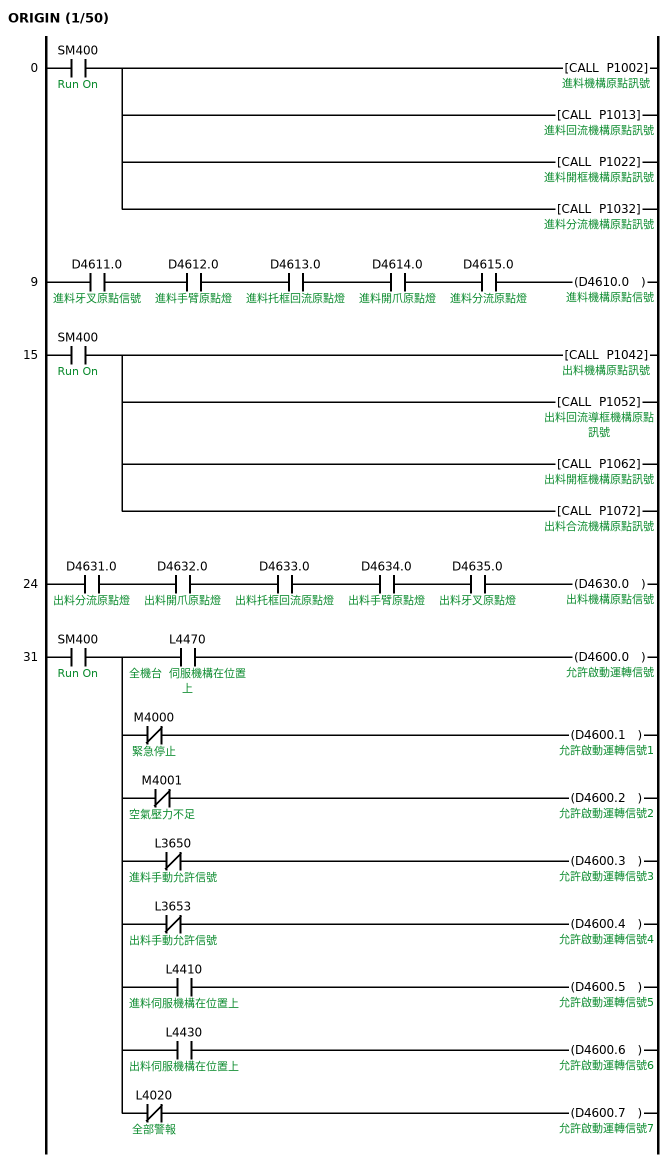
0     LD      SM400  ; Run On
      CALL    P1002  ; 進料機構原點訊號
      CALL    P1013  ; 進料回流機構原點訊號
      CALL    P1022  ; 進料開框機構原點訊號
      CALL    P1032  ; 進料分流機構原點訊號
9     LD      D4611.0  ; 進料牙叉原點信號
      AND     D4612.0  ; 進料手臂原點燈
      AND     D4613.0  ; 進料托框回流原點燈
      AND     D4614.0  ; 進料開爪原點燈
      AND     D4615.0  ; 進料分流原點燈
      OUT     D4610.0  ; 進料機構原點信號
15    LD      SM400  ; Run On
      CALL    P1042  ; 出料機構原點訊號
      CALL    P1052  ; 出料回流導框機構原點訊號
      CALL    P1062  ; 出料開框機構原點訊號
      CALL    P1072  ; 出料合流機構原點訊號
24    LD      D4631.0  ; 出料分流原點燈
      AND     D4632.0  ; 出料開爪原點燈
      AND     D4633.0  ; 出料托框回流原點燈
      AND     D4634.0  ; 出料手臂原點燈
      AND     D4635.0  ; 出料牙叉原點燈
      OUT     D4630.0  ; 出料機構原點信號
31    LD      SM400  ; Run On
      MPS
      AND     L4470  ; 全機台  伺服機構在位置上
      OUT     D4600.0  ; 允許啟動運轉信號
      MRD
      ANI     M4000  ; 緊急停止
      OUT     D4600.1  ; 允許啟動運轉信號1
      MRD
      ANI     M4001  ; 空氣壓力不足
      OUT     D4600.2  ; 允許啟動運轉信號2
      MRD
      ANI     L3650  ; 進料手動允許信號
      OUT     D4600.3  ; 允許啟動運轉信號3
      MRD
      ANI     L3653  ; 出料手動允許信號
      OUT     D4600.4  ; 允許啟動運轉信號4
      MRD
      AND     L4410  ; 進料伺服機構在位置上
      OUT     D4600.5  ; 允許啟動運轉信號5
      MRD
      AND     L4430  ; 出料伺服機構在位置上
      OUT     D4600.6  ; 允許啟動運轉信號6
      MPP
      ANI     L4020  ; 全部警報
      OUT     D4600.7  ; 允許啟動運轉信號7
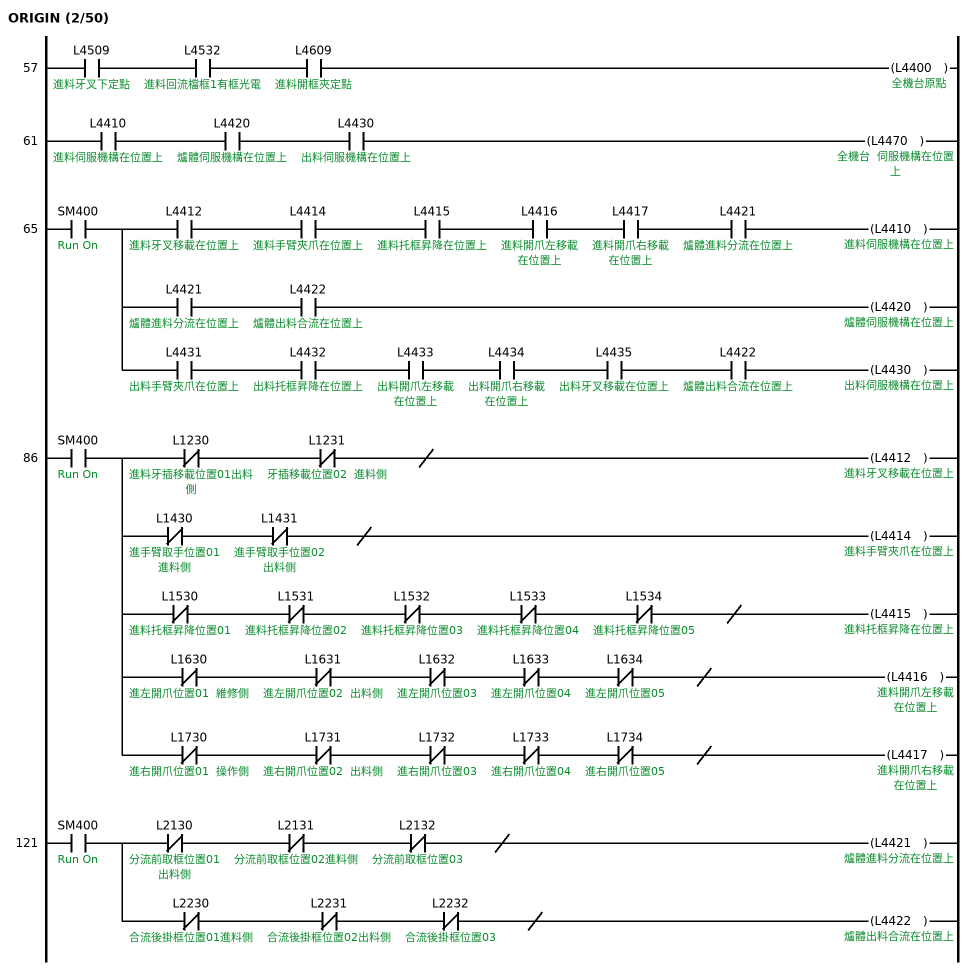
57    LD      L4509  ; 進料牙叉下定點
      AND     L4532  ; 進料回流檔框1有框光電
      AND     L4609  ; 進料開框夾定點
      OUT     L4400  ; 全機台原點
61    LD      L4410  ; 進料伺服機構在位置上
      AND     L4420  ; 爐體伺服機構在位置上
      AND     L4430  ; 出料伺服機構在位置上
      OUT     L4470  ; 全機台  伺服機構在位置上
65    LD      SM400  ; Run On
      MPS
      AND     L4412  ; 進料牙叉移載在位置上
      AND     L4414  ; 進料手臂夾爪在位置上
      AND     L4415  ; 進料托框昇降在位置上
      AND     L4416  ; 進料開爪左移載  在位置上
      AND     L4417  ; 進料開爪右移載  在位置上
      AND     L4421  ; 爐體進料分流在位置上
      OUT     L4410  ; 進料伺服機構在位置上
      MRD
      AND     L4421  ; 爐體進料分流在位置上
      AND     L4422  ; 爐體出料合流在位置上
      OUT     L4420  ; 爐體伺服機構在位置上
      MPP
      AND     L4431  ; 出料手臂夾爪在位置上
      AND     L4432  ; 出料托框昇降在位置上
      AND     L4433  ; 出料開爪左移載  在位置上
      AND     L4434  ; 出料開爪右移載  在位置上
      AND     L4435  ; 出料牙叉移載在位置上
      AND     L4422  ; 爐體出料合流在位置上
      OUT     L4430  ; 出料伺服機構在位置上
86    LD      SM400  ; Run On
      MPS
      ANI     L1230  ; 進料牙插移載位置01出料側
      ANI     L1231  ; 牙插移載位置02  進料側
      INV
      OUT     L4412  ; 進料牙叉移載在位置上
      MRD
      ANI     L1430  ; 進手臂取手位置01  進料側
      ANI     L1431  ; 進手臂取手位置02  出料側
      INV
      OUT     L4414  ; 進料手臂夾爪在位置上
      MRD
      ANI     L1530  ; 進料托框昇降位置01
      ANI     L1531  ; 進料托框昇降位置02
      ANI     L1532  ; 進料托框昇降位置03
      ANI     L1533  ; 進料托框昇降位置04
      ANI     L1534  ; 進料托框昇降位置05
      INV
      OUT     L4415  ; 進料托框昇降在位置上
      MRD
      ANI     L1630  ; 進左開爪位置01  維修側
      ANI     L1631  ; 進左開爪位置02  出料側
      ANI     L1632  ; 進左開爪位置03
      ANI     L1633  ; 進左開爪位置04
      ANI     L1634  ; 進左開爪位置05
      INV
      OUT     L4416  ; 進料開爪左移載  在位置上
      MPP
      ANI     L1730  ; 進右開爪位置01  操作側
      ANI     L1731  ; 進右開爪位置02  出料側
      ANI     L1732  ; 進右開爪位置03
      ANI     L1733  ; 進右開爪位置04
      ANI     L1734  ; 進右開爪位置05
      INV
      OUT     L4417  ; 進料開爪右移載  在位置上
121   LD      SM400  ; Run On
      MPS
      ANI     L2130  ; 分流前取框位置01  出料側
      ANI     L2131  ; 分流前取框位置02進料側
      ANI     L2132  ; 分流前取框位置03
      INV
      OUT     L4421  ; 爐體進料分流在位置上
      MPP
      ANI     L2230  ; 合流後掛框位置01進料側
      ANI     L2231  ; 合流後掛框位置02出料側
      ANI     L2232  ; 合流後掛框位置03
      INV
      OUT     L4422  ; 爐體出料合流在位置上
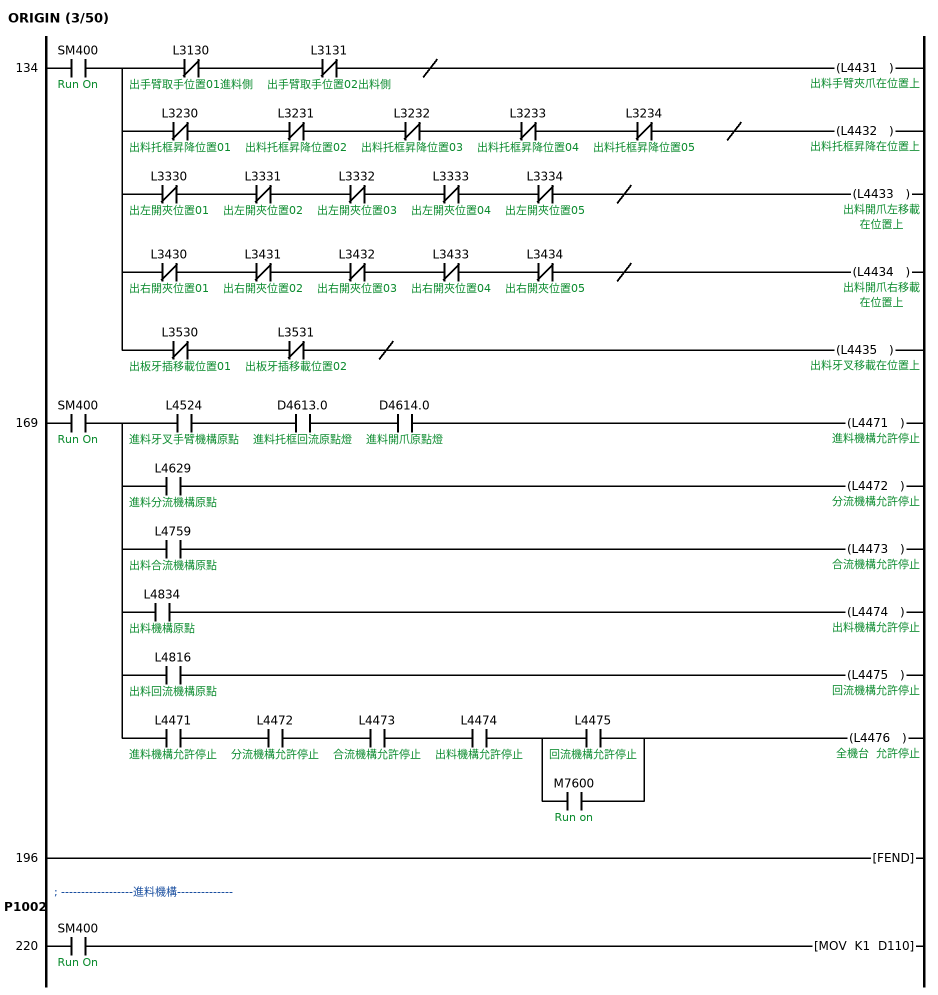
134   LD      SM400  ; Run On
      MPS
      ANI     L3130  ; 出手臂取手位置01進料側
      ANI     L3131  ; 出手臂取手位置02出料側
      INV
      OUT     L4431  ; 出料手臂夾爪在位置上
      MRD
      ANI     L3230  ; 出料托框昇降位置01
      ANI     L3231  ; 出料托框昇降位置02
      ANI     L3232  ; 出料托框昇降位置03
      ANI     L3233  ; 出料托框昇降位置04
      ANI     L3234  ; 出料托框昇降位置05
      INV
      OUT     L4432  ; 出料托框昇降在位置上
      MRD
      ANI     L3330  ; 出左開夾位置01
      ANI     L3331  ; 出左開夾位置02
      ANI     L3332  ; 出左開夾位置03
      ANI     L3333  ; 出左開夾位置04
      ANI     L3334  ; 出左開夾位置05
      INV
      OUT     L4433  ; 出料開爪左移載  在位置上
      MRD
      ANI     L3430  ; 出右開夾位置01
      ANI     L3431  ; 出右開夾位置02
      ANI     L3432  ; 出右開夾位置03
      ANI     L3433  ; 出右開夾位置04
      ANI     L3434  ; 出右開夾位置05
      INV
      OUT     L4434  ; 出料開爪右移載  在位置上
      MPP
      ANI     L3530  ; 出板牙插移載位置01
      ANI     L3531  ; 出板牙插移載位置02
      INV
      OUT     L4435  ; 出料牙叉移載在位置上
169   LD      SM400  ; Run On
      MPS
      AND     L4524  ; 進料牙叉手臂機構原點
      AND     D4613.0  ; 進料托框回流原點燈
      AND     D4614.0  ; 進料開爪原點燈
      OUT     L4471  ; 進料機構允許停止
      MRD
      AND     L4629  ; 進料分流機構原點
      OUT     L4472  ; 分流機構允許停止
      MRD
      AND     L4759  ; 出料合流機構原點
      OUT     L4473  ; 合流機構允許停止
      MRD
      AND     L4834  ; 出料機構原點
      OUT     L4474  ; 出料機構允許停止
      MRD
      AND     L4816  ; 出料回流機構原點
      OUT     L4475  ; 回流機構允許停止
      MPP
      AND     L4471  ; 進料機構允許停止
      AND     L4472  ; 分流機構允許停止
      AND     L4473  ; 合流機構允許停止
      AND     L4474  ; 出料機構允許停止
      LD      L4475  ; 回流機構允許停止
      OR      M7600  ; Run on
      ANB
      OUT     L4476  ; 全機台  允許停止
196   FEND
; ------------------進料機構--------------
      P1002
220   LD      SM400  ; Run On
      MOV     K1 D110
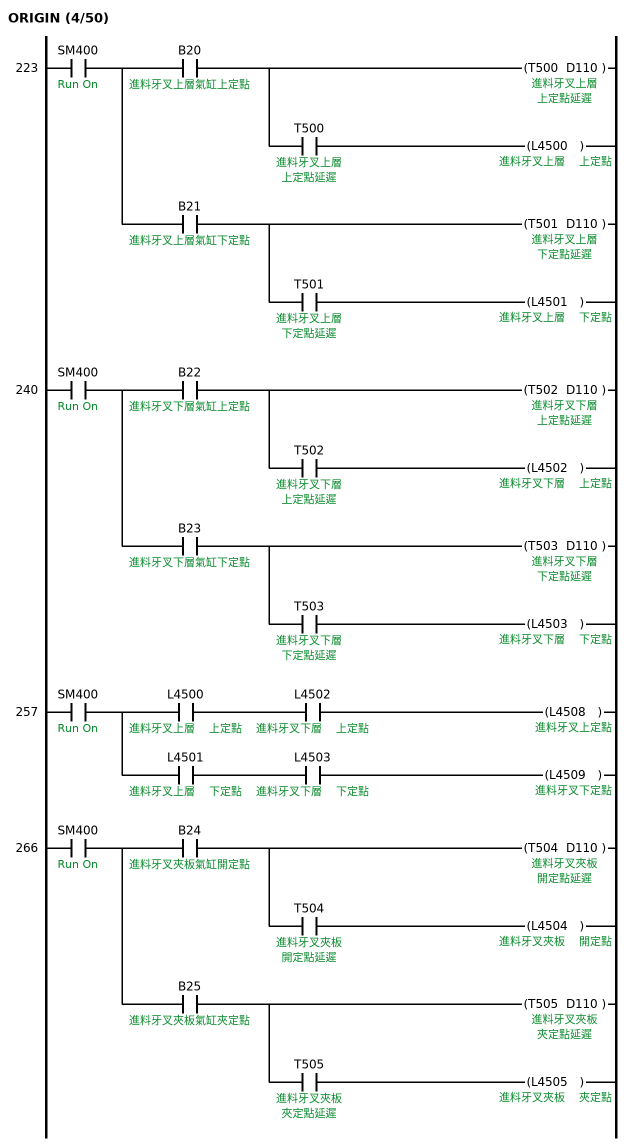
223   LD      SM400  ; Run On
      MPS
      AND     B20  ; 進料牙叉上層氣缸上定點
      OUT     T500 D110  ; 進料牙叉上層    上定點延遲
      AND     T500  ; 進料牙叉上層    上定點延遲
      OUT     L4500  ; 進料牙叉上層    上定點
      MPP
      AND     B21  ; 進料牙叉上層氣缸下定點
      OUT     T501 D110  ; 進料牙叉上層    下定點延遲
      AND     T501  ; 進料牙叉上層    下定點延遲
      OUT     L4501  ; 進料牙叉上層    下定點
240   LD      SM400  ; Run On
      MPS
      AND     B22  ; 進料牙叉下層氣缸上定點
      OUT     T502 D110  ; 進料牙叉下層    上定點延遲
      AND     T502  ; 進料牙叉下層    上定點延遲
      OUT     L4502  ; 進料牙叉下層    上定點
      MPP
      AND     B23  ; 進料牙叉下層氣缸下定點
      OUT     T503 D110  ; 進料牙叉下層    下定點延遲
      AND     T503  ; 進料牙叉下層    下定點延遲
      OUT     L4503  ; 進料牙叉下層    下定點
257   LD      SM400  ; Run On
      MPS
      AND     L4500  ; 進料牙叉上層    上定點
      AND     L4502  ; 進料牙叉下層    上定點
      OUT     L4508  ; 進料牙叉上定點
      MPP
      AND     L4501  ; 進料牙叉上層    下定點
      AND     L4503  ; 進料牙叉下層    下定點
      OUT     L4509  ; 進料牙叉下定點
266   LD      SM400  ; Run On
      MPS
      AND     B24  ; 進料牙叉夾板氣缸開定點
      OUT     T504 D110  ; 進料牙叉夾板    開定點延遲
      AND     T504  ; 進料牙叉夾板    開定點延遲
      OUT     L4504  ; 進料牙叉夾板    開定點
      MPP
      AND     B25  ; 進料牙叉夾板氣缸夾定點
      OUT     T505 D110  ; 進料牙叉夾板    夾定點延遲
      AND     T505  ; 進料牙叉夾板    夾定點延遲
      OUT     L4505  ; 進料牙叉夾板    夾定點
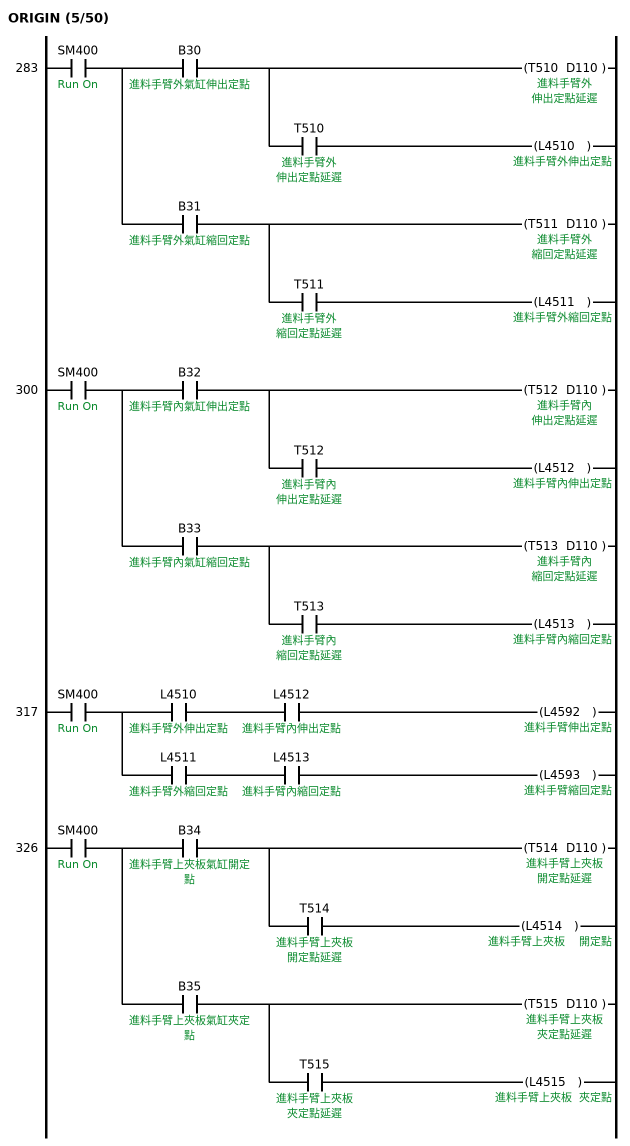
283   LD      SM400  ; Run On
      MPS
      AND     B30  ; 進料手臂外氣缸伸出定點
      OUT     T510 D110  ; 進料手臂外    伸出定點延遲
      AND     T510  ; 進料手臂外    伸出定點延遲
      OUT     L4510  ; 進料手臂外伸出定點
      MPP
      AND     B31  ; 進料手臂外氣缸縮回定點
      OUT     T511 D110  ; 進料手臂外    縮回定點延遲
      AND     T511  ; 進料手臂外    縮回定點延遲
      OUT     L4511  ; 進料手臂外縮回定點
300   LD      SM400  ; Run On
      MPS
      AND     B32  ; 進料手臂內氣缸伸出定點
      OUT     T512 D110  ; 進料手臂內    伸出定點延遲
      AND     T512  ; 進料手臂內    伸出定點延遲
      OUT     L4512  ; 進料手臂內伸出定點
      MPP
      AND     B33  ; 進料手臂內氣缸縮回定點
      OUT     T513 D110  ; 進料手臂內    縮回定點延遲
      AND     T513  ; 進料手臂內    縮回定點延遲
      OUT     L4513  ; 進料手臂內縮回定點
317   LD      SM400  ; Run On
      MPS
      AND     L4510  ; 進料手臂外伸出定點
      AND     L4512  ; 進料手臂內伸出定點
      OUT     L4592  ; 進料手臂伸出定點
      MPP
      AND     L4511  ; 進料手臂外縮回定點
      AND     L4513  ; 進料手臂內縮回定點
      OUT     L4593  ; 進料手臂縮回定點
326   LD      SM400  ; Run On
      MPS
      AND     B34  ; 進料手臂上夾板氣缸開定點
      OUT     T514 D110  ; 進料手臂上夾板    開定點延遲
      AND     T514  ; 進料手臂上夾板    開定點延遲
      OUT     L4514  ; 進料手臂上夾板    開定點
      MPP
      AND     B35  ; 進料手臂上夾板氣缸夾定點
      OUT     T515 D110  ; 進料手臂上夾板    夾定點延遲
      AND     T515  ; 進料手臂上夾板    夾定點延遲
      OUT     L4515  ; 進料手臂上夾板  夾定點
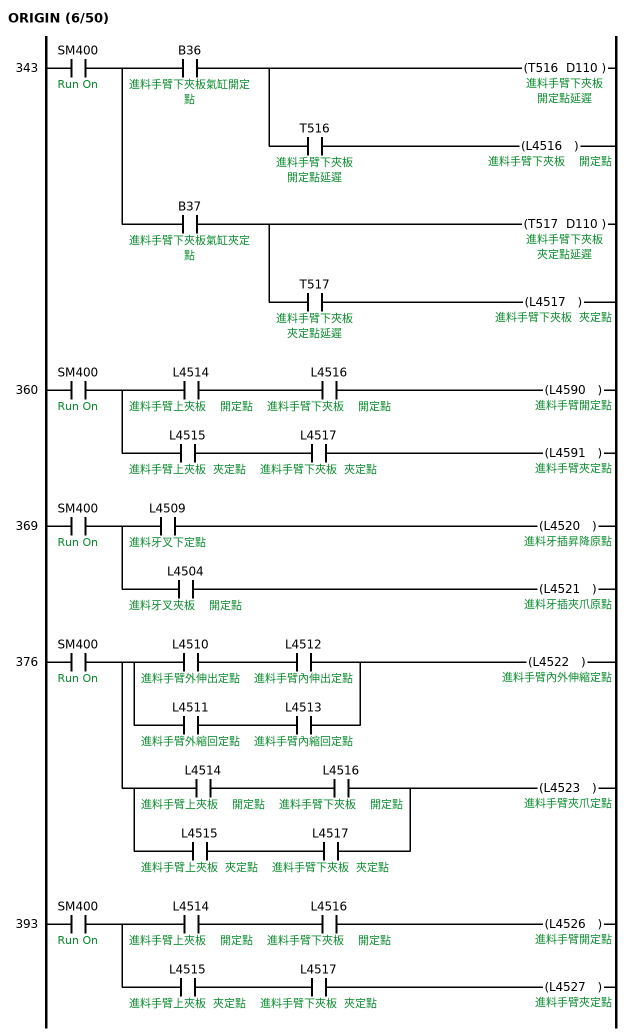
343   LD      SM400  ; Run On
      MPS
      AND     B36  ; 進料手臂下夾板氣缸開定點
      OUT     T516 D110  ; 進料手臂下夾板    開定點延遲
      AND     T516  ; 進料手臂下夾板    開定點延遲
      OUT     L4516  ; 進料手臂下夾板    開定點
      MPP
      AND     B37  ; 進料手臂下夾板氣缸夾定點
      OUT     T517 D110  ; 進料手臂下夾板    夾定點延遲
      AND     T517  ; 進料手臂下夾板    夾定點延遲
      OUT     L4517  ; 進料手臂下夾板  夾定點
360   LD      SM400  ; Run On
      MPS
      AND     L4514  ; 進料手臂上夾板    開定點
      AND     L4516  ; 進料手臂下夾板    開定點
      OUT     L4590  ; 進料手臂開定點
      MPP
      AND     L4515  ; 進料手臂上夾板  夾定點
      AND     L4517  ; 進料手臂下夾板  夾定點
      OUT     L4591  ; 進料手臂夾定點
369   LD      SM400  ; Run On
      MPS
      AND     L4509  ; 進料牙叉下定點
      OUT     L4520  ; 進料牙插昇降原點
      MPP
      AND     L4504  ; 進料牙叉夾板    開定點
      OUT     L4521  ; 進料牙插夾爪原點
376   LD      SM400  ; Run On
      MPS
      LD      L4510  ; 進料手臂外伸出定點
      AND     L4512  ; 進料手臂內伸出定點
      LD      L4511  ; 進料手臂外縮回定點
      AND     L4513  ; 進料手臂內縮回定點
      ORB
      ANB
      OUT     L4522  ; 進料手臂內外伸縮定點
      MPP
      LD      L4514  ; 進料手臂上夾板    開定點
      AND     L4516  ; 進料手臂下夾板    開定點
      LD      L4515  ; 進料手臂上夾板  夾定點
      AND     L4517  ; 進料手臂下夾板  夾定點
      ORB
      ANB
      OUT     L4523  ; 進料手臂夾爪定點
393   LD      SM400  ; Run On
      MPS
      AND     L4514  ; 進料手臂上夾板    開定點
      AND     L4516  ; 進料手臂下夾板    開定點
      OUT     L4526  ; 進料手臂開定點
      MPP
      AND     L4515  ; 進料手臂上夾板  夾定點
      AND     L4517  ; 進料手臂下夾板  夾定點
      OUT     L4527  ; 進料手臂夾定點
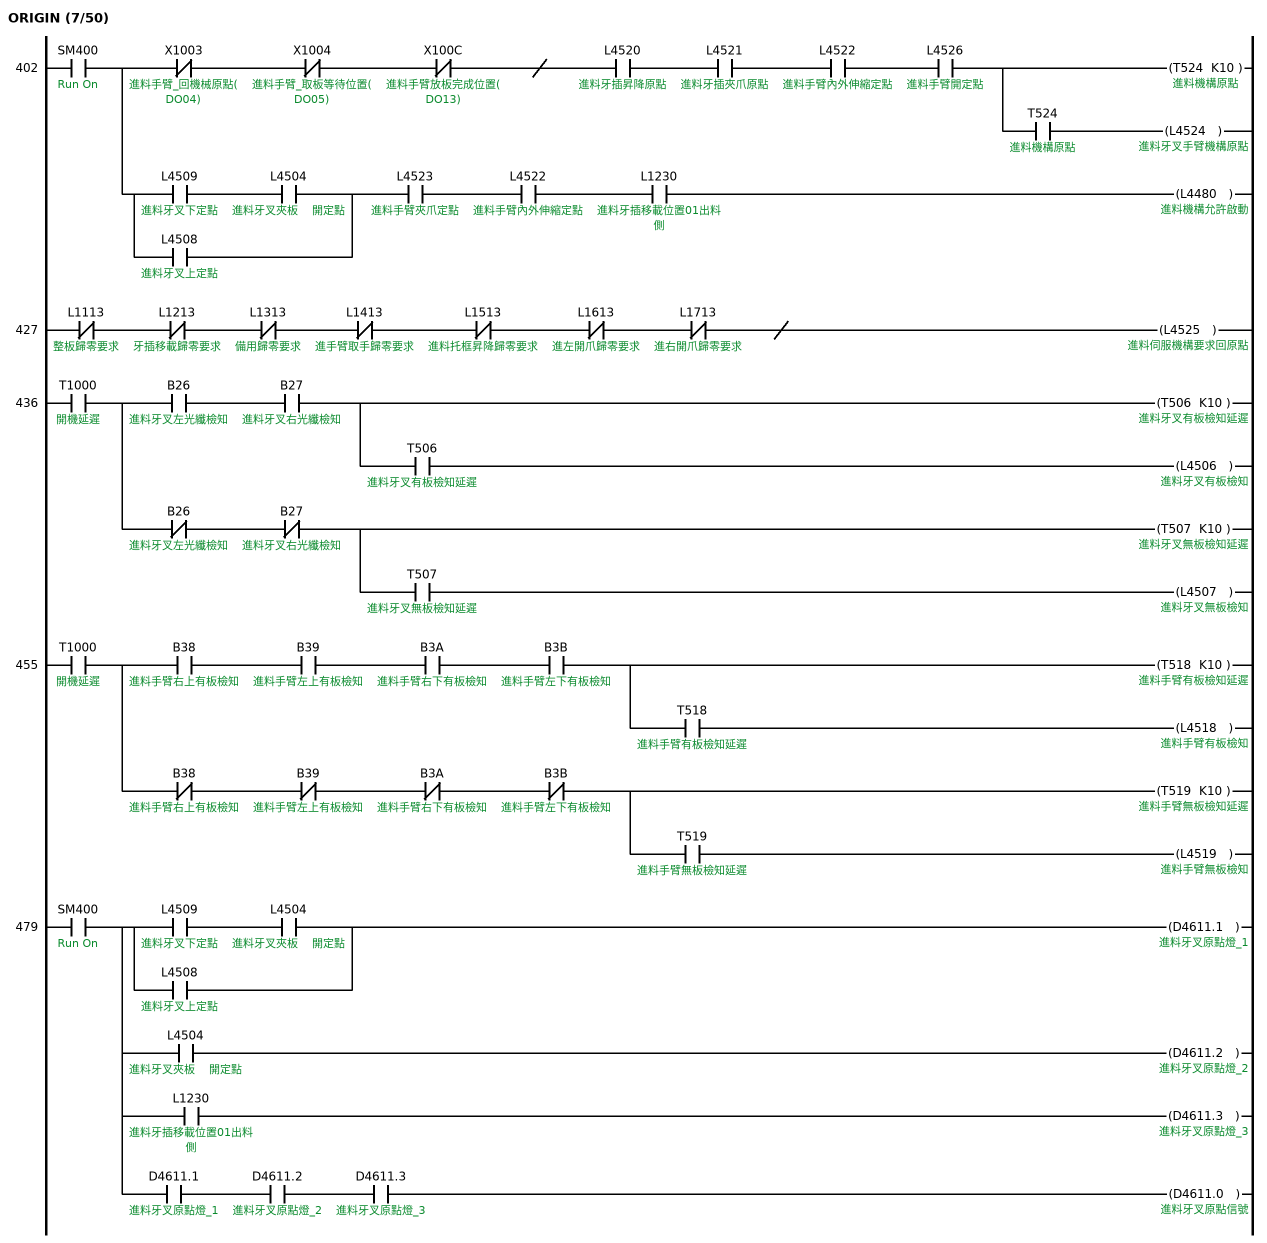
402   LD      SM400  ; Run On
      MPS
      ANI     X1003  ; 進料手臂_回機械原點(DO04)
      ANI     X1004  ; 進料手臂_取板等待位置(DO05)
      ANI     X100C  ; 進料手臂放板完成位置(DO13)
      INV
      AND     L4520  ; 進料牙插昇降原點
      AND     L4521  ; 進料牙插夾爪原點
      AND     L4522  ; 進料手臂內外伸縮定點
      AND     L4526  ; 進料手臂開定點
      OUT     T524 K10  ; 進料機構原點
      AND     T524  ; 進料機構原點
      OUT     L4524  ; 進料牙叉手臂機構原點
      MPP
      LD      L4509  ; 進料牙叉下定點
      AND     L4504  ; 進料牙叉夾板    開定點
      OR      L4508  ; 進料牙叉上定點
      ANB
      AND     L4523  ; 進料手臂夾爪定點
      AND     L4522  ; 進料手臂內外伸縮定點
      AND     L1230  ; 進料牙插移載位置01出料側
      OUT     L4480  ; 進料機構允許啟動
427   LDI     L1113  ; 整板歸零要求
      ANI     L1213  ; 牙插移載歸零要求
      ANI     L1313  ; 備用歸零要求
      ANI     L1413  ; 進手臂取手歸零要求
      ANI     L1513  ; 進料托框昇降歸零要求
      ANI     L1613  ; 進左開爪歸零要求
      ANI     L1713  ; 進右開爪歸零要求
      INV
      OUT     L4525  ; 進料伺服機構要求回原點
436   LD      T1000  ; 開機延遲
      MPS
      AND     B26  ; 進料牙叉左光纖檢知
      AND     B27  ; 進料牙叉右光纖檢知
      OUT     T506 K10  ; 進料牙叉有板檢知延遲
      AND     T506  ; 進料牙叉有板檢知延遲
      OUT     L4506  ; 進料牙叉有板檢知
      MPP
      ANI     B26  ; 進料牙叉左光纖檢知
      ANI     B27  ; 進料牙叉右光纖檢知
      OUT     T507 K10  ; 進料牙叉無板檢知延遲
      AND     T507  ; 進料牙叉無板檢知延遲
      OUT     L4507  ; 進料牙叉無板檢知
455   LD      T1000  ; 開機延遲
      MPS
      AND     B38  ; 進料手臂右上有板檢知
      AND     B39  ; 進料手臂左上有板檢知
      AND     B3A  ; 進料手臂右下有板檢知
      AND     B3B  ; 進料手臂左下有板檢知
      OUT     T518 K10  ; 進料手臂有板檢知延遲
      AND     T518  ; 進料手臂有板檢知延遲
      OUT     L4518  ; 進料手臂有板檢知
      MPP
      ANI     B38  ; 進料手臂右上有板檢知
      ANI     B39  ; 進料手臂左上有板檢知
      ANI     B3A  ; 進料手臂右下有板檢知
      ANI     B3B  ; 進料手臂左下有板檢知
      OUT     T519 K10  ; 進料手臂無板檢知延遲
      AND     T519  ; 進料手臂無板檢知延遲
      OUT     L4519  ; 進料手臂無板檢知
479   LD      SM400  ; Run On
      MPS
      LD      L4509  ; 進料牙叉下定點
      AND     L4504  ; 進料牙叉夾板    開定點
      OR      L4508  ; 進料牙叉上定點
      ANB
      OUT     D4611.1  ; 進料牙叉原點燈_1
      MRD
      AND     L4504  ; 進料牙叉夾板    開定點
      OUT     D4611.2  ; 進料牙叉原點燈_2
      MRD
      AND     L1230  ; 進料牙插移載位置01出料側
      OUT     D4611.3  ; 進料牙叉原點燈_3
      MPP
      AND     D4611.1  ; 進料牙叉原點燈_1
      AND     D4611.2  ; 進料牙叉原點燈_2
      AND     D4611.3  ; 進料牙叉原點燈_3
      OUT     D4611.0  ; 進料牙叉原點信號
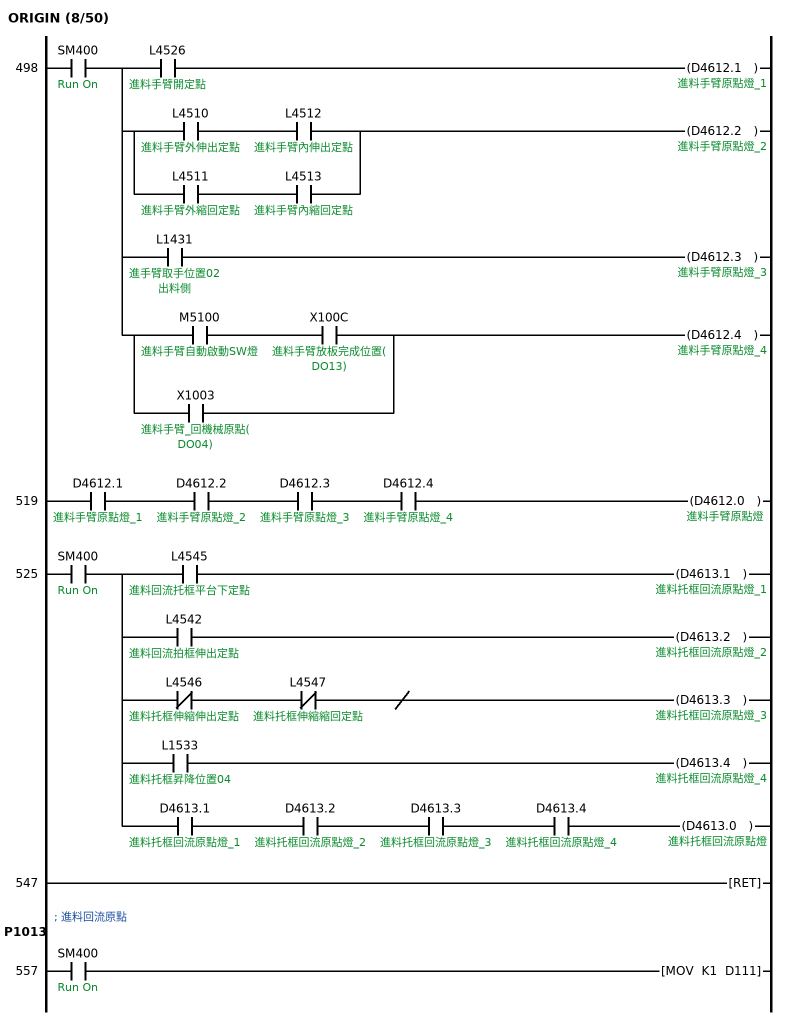
498   LD      SM400  ; Run On
      MPS
      AND     L4526  ; 進料手臂開定點
      OUT     D4612.1  ; 進料手臂原點燈_1
      MRD
      LD      L4510  ; 進料手臂外伸出定點
      AND     L4512  ; 進料手臂內伸出定點
      LD      L4511  ; 進料手臂外縮回定點
      AND     L4513  ; 進料手臂內縮回定點
      ORB
      ANB
      OUT     D4612.2  ; 進料手臂原點燈_2
      MRD
      AND     L1431  ; 進手臂取手位置02  出料側
      OUT     D4612.3  ; 進料手臂原點燈_3
      MPP
      LD      M5100  ; 進料手臂自動啟動SW燈
      AND     X100C  ; 進料手臂放板完成位置(DO13)
      OR      X1003  ; 進料手臂_回機械原點(DO04)
      ANB
      OUT     D4612.4  ; 進料手臂原點燈_4
519   LD      D4612.1  ; 進料手臂原點燈_1
      AND     D4612.2  ; 進料手臂原點燈_2
      AND     D4612.3  ; 進料手臂原點燈_3
      AND     D4612.4  ; 進料手臂原點燈_4
      OUT     D4612.0  ; 進料手臂原點燈
525   LD      SM400  ; Run On
      MPS
      AND     L4545  ; 進料回流托框平台下定點
      OUT     D4613.1  ; 進料托框回流原點燈_1
      MRD
      AND     L4542  ; 進料回流拍框伸出定點
      OUT     D4613.2  ; 進料托框回流原點燈_2
      MRD
      ANI     L4546  ; 進料托框伸縮伸出定點
      ANI     L4547  ; 進料托框伸縮縮回定點
      INV
      OUT     D4613.3  ; 進料托框回流原點燈_3
      MRD
      AND     L1533  ; 進料托框昇降位置04
      OUT     D4613.4  ; 進料托框回流原點燈_4
      MPP
      AND     D4613.1  ; 進料托框回流原點燈_1
      AND     D4613.2  ; 進料托框回流原點燈_2
      AND     D4613.3  ; 進料托框回流原點燈_3
      AND     D4613.4  ; 進料托框回流原點燈_4
      OUT     D4613.0  ; 進料托框回流原點燈
547   RET
; 進料回流原點
      P1013
557   LD      SM400  ; Run On
      MOV     K1 D111
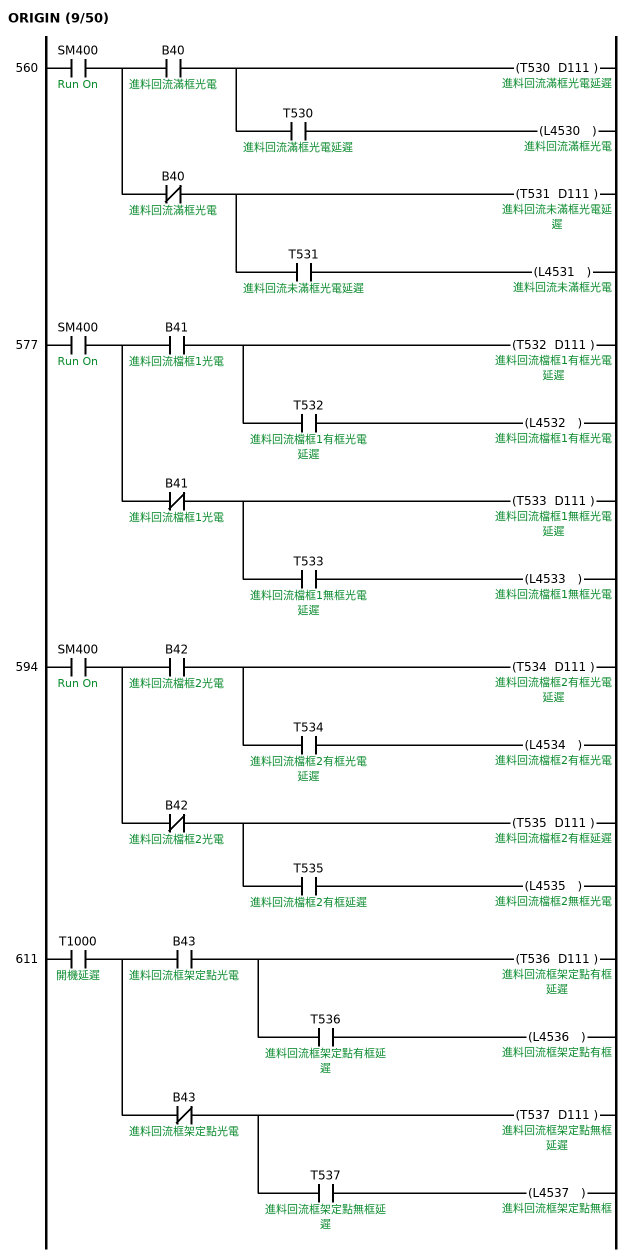
560   LD      SM400  ; Run On
      MPS
      AND     B40  ; 進料回流滿框光電
      OUT     T530 D111  ; 進料回流滿框光電延遲
      AND     T530  ; 進料回流滿框光電延遲
      OUT     L4530  ; 進料回流滿框光電
      MPP
      ANI     B40  ; 進料回流滿框光電
      OUT     T531 D111  ; 進料回流未滿框光電延遲
      AND     T531  ; 進料回流未滿框光電延遲
      OUT     L4531  ; 進料回流未滿框光電
577   LD      SM400  ; Run On
      MPS
      AND     B41  ; 進料回流檔框1光電
      OUT     T532 D111  ; 進料回流檔框1有框光電延遲
      AND     T532  ; 進料回流檔框1有框光電延遲
      OUT     L4532  ; 進料回流檔框1有框光電
      MPP
      ANI     B41  ; 進料回流檔框1光電
      OUT     T533 D111  ; 進料回流檔框1無框光電延遲
      AND     T533  ; 進料回流檔框1無框光電延遲
      OUT     L4533  ; 進料回流檔框1無框光電
594   LD      SM400  ; Run On
      MPS
      AND     B42  ; 進料回流檔框2光電
      OUT     T534 D111  ; 進料回流檔框2有框光電延遲
      AND     T534  ; 進料回流檔框2有框光電延遲
      OUT     L4534  ; 進料回流檔框2有框光電
      MPP
      ANI     B42  ; 進料回流檔框2光電
      OUT     T535 D111  ; 進料回流檔框2有框延遲
      AND     T535  ; 進料回流檔框2有框延遲
      OUT     L4535  ; 進料回流檔框2無框光電
611   LD      T1000  ; 開機延遲
      MPS
      AND     B43  ; 進料回流框架定點光電
      OUT     T536 D111  ; 進料回流框架定點有框延遲
      AND     T536  ; 進料回流框架定點有框延遲
      OUT     L4536  ; 進料回流框架定點有框
      MPP
      ANI     B43  ; 進料回流框架定點光電
      OUT     T537 D111  ; 進料回流框架定點無框延遲
      AND     T537  ; 進料回流框架定點無框延遲
      OUT     L4537  ; 進料回流框架定點無框
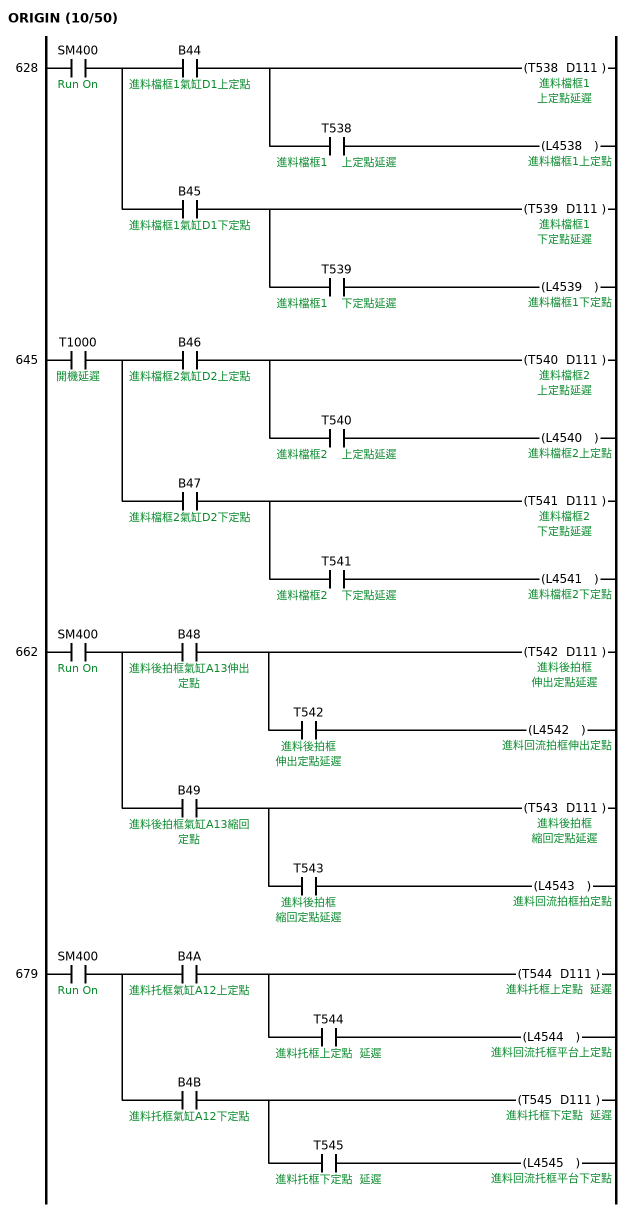
628   LD      SM400  ; Run On
      MPS
      AND     B44  ; 進料檔框1氣缸D1上定點
      OUT     T538 D111  ; 進料檔框1    上定點延遲
      AND     T538  ; 進料檔框1    上定點延遲
      OUT     L4538  ; 進料檔框1上定點
      MPP
      AND     B45  ; 進料檔框1氣缸D1下定點
      OUT     T539 D111  ; 進料檔框1    下定點延遲
      AND     T539  ; 進料檔框1    下定點延遲
      OUT     L4539  ; 進料檔框1下定點
645   LD      T1000  ; 開機延遲
      MPS
      AND     B46  ; 進料檔框2氣缸D2上定點
      OUT     T540 D111  ; 進料檔框2    上定點延遲
      AND     T540  ; 進料檔框2    上定點延遲
      OUT     L4540  ; 進料檔框2上定點
      MPP
      AND     B47  ; 進料檔框2氣缸D2下定點
      OUT     T541 D111  ; 進料檔框2    下定點延遲
      AND     T541  ; 進料檔框2    下定點延遲
      OUT     L4541  ; 進料檔框2下定點
662   LD      SM400  ; Run On
      MPS
      AND     B48  ; 進料後拍框氣缸A13伸出定點
      OUT     T542 D111  ; 進料後拍框    伸出定點延遲
      AND     T542  ; 進料後拍框    伸出定點延遲
      OUT     L4542  ; 進料回流拍框伸出定點
      MPP
      AND     B49  ; 進料後拍框氣缸A13縮回定點
      OUT     T543 D111  ; 進料後拍框    縮回定點延遲
      AND     T543  ; 進料後拍框    縮回定點延遲
      OUT     L4543  ; 進料回流拍框拍定點
679   LD      SM400  ; Run On
      MPS
      AND     B4A  ; 進料托框氣缸A12上定點
      OUT     T544 D111  ; 進料托框上定點  延遲
      AND     T544  ; 進料托框上定點  延遲
      OUT     L4544  ; 進料回流托框平台上定點
      MPP
      AND     B4B  ; 進料托框氣缸A12下定點
      OUT     T545 D111  ; 進料托框下定點  延遲
      AND     T545  ; 進料托框下定點  延遲
      OUT     L4545  ; 進料回流托框平台下定點
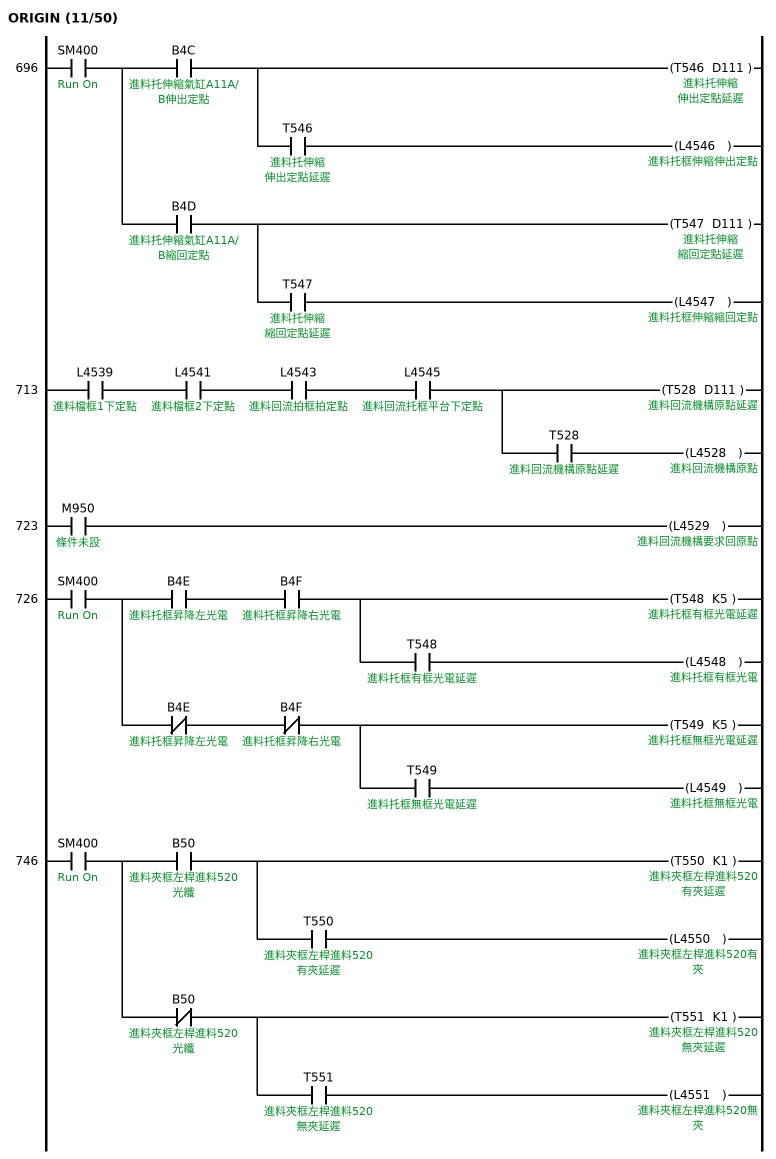
696   LD      SM400  ; Run On
      MPS
      AND     B4C  ; 進料托伸縮氣缸A11A/B伸出定點
      OUT     T546 D111  ; 進料托伸縮    伸出定點延遲
      AND     T546  ; 進料托伸縮    伸出定點延遲
      OUT     L4546  ; 進料托框伸縮伸出定點
      MPP
      AND     B4D  ; 進料托伸縮氣缸A11A/B縮回定點
      OUT     T547 D111  ; 進料托伸縮    縮回定點延遲
      AND     T547  ; 進料托伸縮    縮回定點延遲
      OUT     L4547  ; 進料托框伸縮縮回定點
713   LD      L4539  ; 進料檔框1下定點
      AND     L4541  ; 進料檔框2下定點
      AND     L4543  ; 進料回流拍框拍定點
      AND     L4545  ; 進料回流托框平台下定點
      OUT     T528 D111  ; 進料回流機構原點延遲
      AND     T528  ; 進料回流機構原點延遲
      OUT     L4528  ; 進料回流機構原點
723   LD      M950  ; 條件未設
      OUT     L4529  ; 進料回流機構要求回原點
726   LD      SM400  ; Run On
      MPS
      AND     B4E  ; 進料托框昇降左光電
      AND     B4F  ; 進料托框昇降右光電
      OUT     T548 K5  ; 進料托框有框光電延遲
      AND     T548  ; 進料托框有框光電延遲
      OUT     L4548  ; 進料托框有框光電
      MPP
      ANI     B4E  ; 進料托框昇降左光電
      ANI     B4F  ; 進料托框昇降右光電
      OUT     T549 K5  ; 進料托框無框光電延遲
      AND     T549  ; 進料托框無框光電延遲
      OUT     L4549  ; 進料托框無框光電
746   LD      SM400  ; Run On
      MPS
      AND     B50  ; 進料夾框左桿進料520 光纖
      OUT     T550 K1  ; 進料夾框左桿進料520 有夾延遲
      AND     T550  ; 進料夾框左桿進料520 有夾延遲
      OUT     L4550  ; 進料夾框左桿進料520有夾
      MPP
      ANI     B50  ; 進料夾框左桿進料520 光纖
      OUT     T551 K1  ; 進料夾框左桿進料520 無夾延遲
      AND     T551  ; 進料夾框左桿進料520 無夾延遲
      OUT     L4551  ; 進料夾框左桿進料520無夾
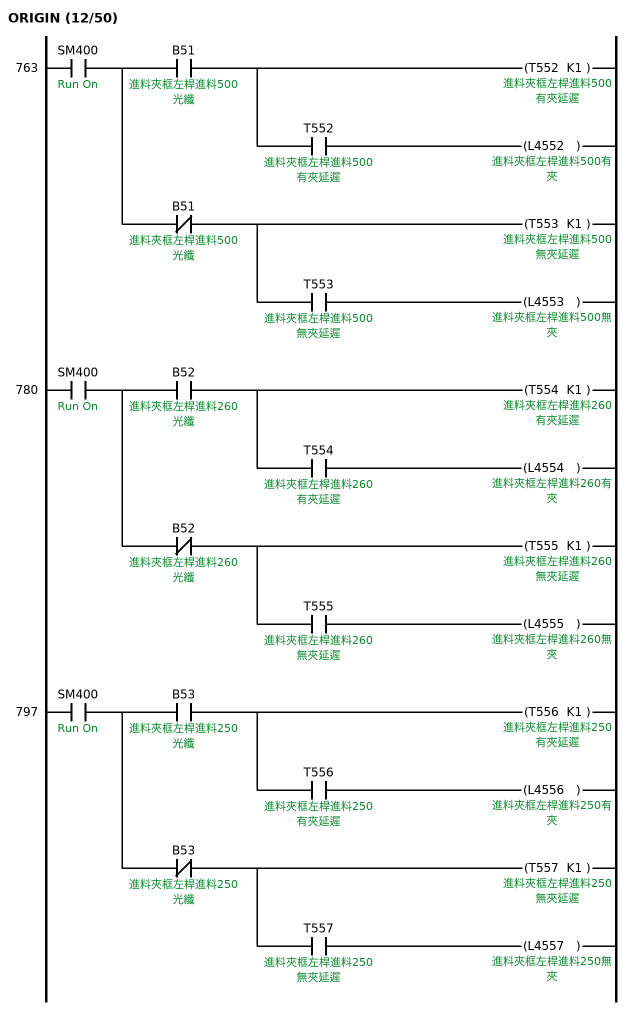
763   LD      SM400  ; Run On
      MPS
      AND     B51  ; 進料夾框左桿進料500 光纖
      OUT     T552 K1  ; 進料夾框左桿進料500 有夾延遲
      AND     T552  ; 進料夾框左桿進料500 有夾延遲
      OUT     L4552  ; 進料夾框左桿進料500有夾
      MPP
      ANI     B51  ; 進料夾框左桿進料500 光纖
      OUT     T553 K1  ; 進料夾框左桿進料500 無夾延遲
      AND     T553  ; 進料夾框左桿進料500 無夾延遲
      OUT     L4553  ; 進料夾框左桿進料500無夾
780   LD      SM400  ; Run On
      MPS
      AND     B52  ; 進料夾框左桿進料260 光纖
      OUT     T554 K1  ; 進料夾框左桿進料260 有夾延遲
      AND     T554  ; 進料夾框左桿進料260 有夾延遲
      OUT     L4554  ; 進料夾框左桿進料260有夾
      MPP
      ANI     B52  ; 進料夾框左桿進料260 光纖
      OUT     T555 K1  ; 進料夾框左桿進料260 無夾延遲
      AND     T555  ; 進料夾框左桿進料260 無夾延遲
      OUT     L4555  ; 進料夾框左桿進料260無夾
797   LD      SM400  ; Run On
      MPS
      AND     B53  ; 進料夾框左桿進料250 光纖
      OUT     T556 K1  ; 進料夾框左桿進料250 有夾延遲
      AND     T556  ; 進料夾框左桿進料250 有夾延遲
      OUT     L4556  ; 進料夾框左桿進料250有夾
      MPP
      ANI     B53  ; 進料夾框左桿進料250 光纖
      OUT     T557 K1  ; 進料夾框左桿進料250 無夾延遲
      AND     T557  ; 進料夾框左桿進料250 無夾延遲
      OUT     L4557  ; 進料夾框左桿進料250無夾
